C09107=1097.158,375.696,407.850,178.891,20.769,152.741
C09108=1097.152,375.448,407.886,178.888,20.763,152.740
C09109=1097.146,375.200,407.923,178.886,20.758,152.739
C09110=1097.140,374.954,407.959,178.883,20.754,152.739
C09111=1097.134,374.706,407.995,178.880,20.748,152.738
C09112=1097.129,374.459,408.032,178.878,20.743,152.737
C09113=1097.123,374.211,408.068,178.875,20.738,152.736
C09114=1097.118,373.965,408.104,178.872,20.733,152.736
C09115=1097.111,373.718,408.141,178.869,20.728,152.735
C09116=1097.105,373.470,408.177,178.866,20.722,152.734
C09117=1097.099,373.223,408.213,178.863,20.718,152.733
C09118=1097.094,372.976,408.249,178.860,20.712,152.733
C09119=1097.088,372.729,408.286,178.857,20.708,152.732
C09120=1097.082,372.481,408.321,178.855,20.703,152.731
C09121=1097.076,372.234,408.358,178.851,20.698,152.730
C09122=1097.070,371.987,408.393,178.849,20.693,152.730
C09123=1097.065,371.739,408.429,178.845,20.688,152.729
C09124=1097.059,371.492,408.466,178.842,20.683,152.728
C09125=1097.053,371.245,408.501,178.839,20.678,152.728
C09126=1097.047,370.998,408.538,178.836,20.673,152.727
C09127=1097.037,370.603,408.595,178.832,20.665,152.726
C09128=1097.029,370.208,408.652,178.828,20.657,152.725
C09129=1097.019,369.813,408.710,178.823,20.649,152.724
C09130=1097.010,369.418,408.767,178.818,20.642,152.722
C09131=1097.004,369.171,408.802,178.816,20.637,152.722
C09132=1096.999,368.924,408.838,178.812,20.632,152.721
C09133=1096.993,368.677,408.874,178.809,20.628,152.721
C09134=1096.987,368.429,408.910,178.806,20.623,152.720
C09135=1096.982,368.182,408.946,178.803,20.617,152.719
C09136=1096.976,367.934,408.982,178.801,20.613,152.718
C09137=1096.970,367.688,409.018,178.798,20.608,152.718
C09138=1096.964,367.440,409.053,178.795,20.603,152.717
C09139=1096.958,367.192,409.089,178.792,20.599,152.716
C09140=1096.953,366.945,409.125,178.789,20.594,152.716
C09141=1096.947,366.698,409.160,178.786,20.589,152.715
C09142=1096.941,366.451,409.196,178.783,20.585,152.715
C09143=1096.935,366.203,409.231,178.780,20.580,152.714
C09144=1096.930,365.956,409.267,178.777,20.575,152.713
C09145=1096.924,365.708,409.302,178.774,20.570,152.713
C09146=1096.918,365.461,409.338,178.772,20.566,152.712
C09147=1096.912,365.214,409.374,178.769,20.561,152.711
C09148=1096.906,364.966,409.409,178.766,20.556,152.711
C09149=1096.901,364.719,409.445,178.762,20.552,152.710
C09150=1096.895,364.471,409.480,178.760,20.548,152.710
C09151=1096.889,364.224,409.516,178.757,20.543,152.709
C09152=1096.884,363.976,409.551,178.754,20.538,152.708
C09153=1096.878,363.729,409.586,178.750,20.534,152.708
C09154=1096.872,363.482,409.622,178.747,20.529,152.707
C09155=1096.866,363.235,409.657,178.745,20.525,152.707
C09156=1096.860,362.987,409.692,178.742,20.520,152.706
C09157=1096.854,362.740,409.728,178.739,20.515,152.705
C09158=1096.849,362.492,409.763,178.736,20.512,152.705
C09159=1096.843,362.245,409.798,178.733,20.507,152.704
C09160=1096.837,361.997,409.834,178.730,20.502,152.704
C09161=1096.831,361.751,409.869,178.727,20.497,152.703
C09162=1096.825,361.502,409.904,178.724,20.494,152.703
C09163=1096.820,361.255,409.939,178.721,20.489,152.702
C09164=1096.814,361.008,409.975,178.718,20.484,152.701
C09165=1096.809,360.760,410.009,178.714,20.480,152.701
C09166=1096.803,360.513,410.044,178.712,20.476,152.700
C09167=1096.797,360.266,410.080,178.709,20.471,152.700
C09168=1096.791,360.018,410.114,178.706,20.467,152.699
C09169=1096.785,359.770,410.150,178.703,20.463,152.699
C09170=1096.780,359.523,410.184,178.700,20.458,152.698
C09171=1096.774,359.276,410.220,178.697,20.453,152.698
C09172=1096.768,359.029,410.255,178.694,20.450,152.697
C09173=1096.762,358.781,410.290,178.691,20.445,152.697
C09174=1096.756,358.534,410.325,178.688,20.441,152.696
C09175=1096.750,358.286,410.359,178.685,20.437,152.696
C09176=1096.744,358.039,410.395,178.682,20.432,152.695
C09177=1096.739,357.791,410.430,178.679,20.428,152.695
C09178=1096.732,357.544,410.465,178.676,20.424,152.694
C09179=1096.724,357.164,410.517,178.671,20.417,152.693
C09180=1096.716,356.784,410.572,178.667,20.410,152.692
C09181=1096.707,356.405,410.625,178.662,20.404,152.692
C09182=1096.698,356.025,410.678,178.658,20.398,152.691
C09183=1096.692,355.778,410.713,178.654,20.393,152.690
C09184=1096.686,355.530,410.748,178.652,20.389,152.690
C09185=1096.681,355.282,410.782,178.648,20.385,152.689
C09186=1096.675,355.035,410.817,178.645,20.381,152.689
C09187=1096.669,354.787,410.852,178.643,20.377,152.688
C09188=1096.663,354.540,410.886,178.639,20.372,152.688
C09189=1096.658,354.292,410.921,178.637,20.369,152.687
C09190=1096.652,354.044,410.955,178.634,20.364,152.687
C09191=1096.646,353.797,410.991,178.630,20.360,152.687
C09192=1096.640,353.550,411.025,178.628,20.356,152.686
C09193=1096.635,353.302,411.059,178.624,20.352,152.686
C09194=1096.629,353.054,411.094,178.621,20.348,152.685
C09195=1096.624,352.807,411.128,178.618,20.344,152.685
C09196=1096.618,352.560,411.162,178.615,20.339,152.684
C09197=1096.611,352.312,411.197,178.612,20.336,152.684
C09198=1096.606,352.065,411.232,178.609,20.331,152.683
C09199=1096.600,351.817,411.266,178.606,20.328,152.683
C09200=1096.594,351.570,411.300,178.603,20.324,152.682
C09201=1096.588,351.322,411.335,178.600,20.320,152.682
C09202=1096.583,351.074,411.369,178.597,20.316,152.682
C09203=1096.577,350.827,411.403,178.594,20.312,152.681
C09204=1096.572,350.580,411.438,178.591,20.308,152.681
C09205=1096.565,350.332,411.473,178.588,20.304,152.680
C09206=1096.559,350.084,411.507,178.584,20.299,152.680
C09207=1096.554,349.837,411.541,178.582,20.296,152.679
C09208=1096.549,349.589,411.575,178.578,20.292,152.679
C09209=1096.542,349.341,411.609,178.576,20.288,152.679
C09210=1096.537,349.093,411.644,178.572,20.284,152.678
C09211=1096.531,348.846,411.678,178.570,20.280,152.678
C09212=1096.525,348.599,411.712,178.566,20.276,152.677
C09213=1096.519,348.351,411.746,178.564,20.273,152.677
C09214=1096.514,348.103,411.781,178.560,20.269,152.677
C09215=1096.508,347.855,411.814,178.557,20.264,152.676
C09216=1096.502,347.608,411.848,178.554,20.261,152.676
C09217=1096.496,347.361,411.882,178.551,20.257,152.675
C09218=1096.491,347.113,411.917,178.548,20.253,152.675
C09219=1096.486,346.865,411.950,178.545,20.249,152.675
C09220=1096.480,346.618,411.984,178.542,20.245,152.674
C09221=1096.473,346.370,412.019,178.539,20.241,152.674
C09222=1096.468,346.123,412.053,178.536,20.238,152.673
C09223=1096.463,345.874,412.087,178.532,20.234,152.673
C09224=1096.457,345.627,412.121,178.530,20.230,152.673
C09225=1096.451,345.379,412.154,178.527,20.226,152.672
C09226=1096.445,345.132,412.188,178.524,20.222,152.672
C09227=1096.440,344.885,412.222,178.520,20.218,152.671
C09228=1096.434,344.637,412.256,178.518,20.215,152.671
C09229=1096.428,344.389,412.290,178.514,20.211,152.671
C09230=1096.422,344.141,412.323,178.512,20.207,152.670
C09231=1096.413,343.764,412.375,178.507,20.202,152.670
C09232=1096.405,343.387,412.427,178.502,20.196,152.669
C09233=1096.396,343.009,412.478,178.497,20.190,152.669
C09234=1096.387,342.632,412.529,178.492,20.185,152.668
C09235=1096.381,342.385,412.563,178.489,20.181,152.668
C09236=1096.376,342.137,412.596,178.487,20.178,152.668
C09237=1096.370,341.890,412.630,178.483,20.174,152.667
C09238=1096.365,341.642,412.664,178.481,20.170,152.667
C09239=1096.359,341.394,412.698,178.477,20.167,152.667
C09240=1096.353,341.147,412.731,178.474,20.163,152.666
C09241=1096.347,340.898,412.765,178.471,20.159,152.666
C09242=1096.341,340.651,412.799,178.468,20.156,152.666
C09243=1096.336,340.403,412.832,178.465,20.152,152.665
C09244=1096.330,340.155,412.865,178.462,20.149,152.665
C09245=1096.324,339.907,412.899,178.458,20.145,152.665
C09246=1096.318,339.660,412.932,178.455,20.141,152.664
C09247=1096.312,339.412,412.966,178.453,20.138,152.664
C09248=1096.307,339.165,412.999,178.449,20.134,152.664
C09249=1096.302,338.917,413.032,178.446,20.131,152.663
C09250=1096.296,338.670,413.066,178.443,20.127,152.663
C09251=1096.290,338.422,413.099,178.440,20.124,152.663
C09252=1096.285,338.174,413.133,178.437,20.120,152.662
C09253=1096.278,337.926,413.165,178.434,20.116,152.662
C09254=1096.273,337.678,413.199,178.431,20.113,152.662
C09255=1096.267,337.430,413.232,178.427,20.109,152.662
C09256=1096.262,337.183,413.266,178.425,20.106,152.661
C09257=1096.255,336.936,413.299,178.421,20.102,152.661
C09258=1096.250,336.688,413.332,178.418,20.099,152.661
C09259=1096.244,336.440,413.365,178.415,20.096,152.660
C09260=1096.239,336.192,413.399,178.412,20.092,152.660
C09261=1096.232,335.944,413.432,178.409,20.089,152.660
C09262=1096.227,335.696,413.465,178.405,20.085,152.660
C09263=1096.221,335.448,413.498,178.403,20.082,152.659
C09264=1096.215,335.201,413.531,178.400,20.079,152.659
C09265=1096.209,334.953,413.564,178.396,20.075,152.659
C09266=1096.204,334.705,413.598,178.393,20.072,152.658
C09267=1096.198,334.457,413.631,178.391,20.069,152.658
C09268=1096.193,334.210,413.663,178.387,20.064,152.658
C09269=1096.187,333.962,413.697,178.384,20.061,152.658
C09270=1096.181,333.714,413.730,178.382,20.058,152.657
C09271=1096.175,333.466,413.762,178.378,20.054,152.657
C09272=1096.170,333.218,413.795,178.375,20.051,152.657
C09273=1096.164,332.971,413.828,178.371,20.047,152.657
C09274=1096.158,332.723,413.861,178.369,20.044,152.656
C09275=1096.153,332.476,413.894,178.366,20.041,152.656
C09276=1096.147,332.228,413.927,178.362,20.038,152.656
C09277=1096.142,331.979,413.960,178.359,20.034,152.656
C09278=1096.135,331.732,413.993,178.356,20.031,152.655
C09279=1096.130,331.484,414.026,178.353,20.027,152.655
C09280=1096.123,331.236,414.059,178.350,20.024,152.655
C09281=1096.118,330.988,414.091,178.347,20.021,152.655
C09282=1096.112,330.740,414.124,178.343,20.018,152.654
C09283=1096.103,330.358,414.174,178.339,20.013,152.654
C09284=1096.094,329.974,414.225,178.334,20.008,152.654
C09285=1096.085,329.591,414.276,178.329,20.003,152.653
C09286=1096.076,329.208,414.326,178.324,19.998,152.653
C09287=1096.070,328.960,414.359,178.321,19.995,152.653
C09288=1096.064,328.712,414.391,178.318,19.992,152.653
C09289=1096.059,328.464,414.424,178.315,19.989,152.653
C09290=1096.053,328.216,414.456,178.312,19.986,152.652
C09291=1096.047,327.969,414.489,178.308,19.982,152.652
C09292=1096.042,327.721,414.521,178.305,19.979,152.652
C09293=1096.035,327.473,414.554,178.303,19.976,152.652
C09294=1096.029,327.225,414.586,178.299,19.973,152.652
C09295=1096.024,326.978,414.619,178.296,19.970,152.651
C09296=1096.019,326.729,414.651,178.293,19.967,152.651
C09297=1096.012,326.482,414.684,178.290,19.964,152.651
C09298=1096.006,326.234,414.716,178.286,19.960,152.651
C09299=1096.001,325.986,414.749,178.283,19.957,152.651
C09300=1095.995,325.738,414.781,178.281,19.954,152.650
C09301=1095.989,325.491,414.814,178.278,19.951,152.650
C09302=1095.983,325.242,414.846,178.274,19.948,152.650
C09303=1095.978,324.994,414.878,178.271,19.945,152.650
C09304=1095.972,324.747,414.911,178.268,19.942,152.650
C09305=1095.966,324.499,414.943,178.265,19.939,152.649
C09306=1095.961,324.251,414.974,178.261,19.935,152.649
C09307=1095.955,324.003,415.008,178.258,19.932,152.649
C09308=1095.949,323.755,415.040,178.255,19.929,152.649
C09309=1095.944,323.508,415.071,178.253,19.926,152.649
C09310=1095.938,323.259,415.103,178.249,19.923,152.648
C09311=1095.933,323.012,415.136,178.246,19.920,152.648
C09312=1095.927,322.764,415.168,178.243,19.917,152.648
C09313=1095.921,322.516,415.200,178.240,19.914,152.648
C09314=1095.915,322.268,415.232,178.236,19.910,152.648
C09315=1095.909,322.020,415.264,178.233,19.908,152.648
C09316=1095.903,321.772,415.297,178.230,19.905,152.647
C09317=1095.899,321.525,415.329,178.227,19.902,152.647
C09318=1095.893,321.276,415.361,178.223,19.899,152.647
C09319=1095.887,321.029,415.393,178.221,19.895,152.647
C09320=1095.881,320.781,415.425,178.218,19.892,152.647
C09321=1095.876,320.533,415.457,178.215,19.890,152.647
C09322=1095.870,320.285,415.489,178.212,19.887,152.646
C09323=1095.864,320.037,415.520,178.208,19.883,152.646
C09324=1095.859,319.789,415.554,178.205,19.881,152.646
C09325=1095.853,319.541,415.586,178.202,19.877,152.646
C09326=1095.848,319.294,415.617,178.199,19.874,152.646
C09327=1095.842,319.046,415.649,178.196,19.872,152.646
C09328=1095.836,318.798,415.681,178.192,19.868,152.645
C09329=1095.830,318.550,415.713,178.190,19.865,152.645
C09330=1095.825,318.302,415.745,178.186,19.863,152.645
C09331=1095.820,318.054,415.776,178.184,19.860,152.645
C09332=1095.814,317.806,415.808,178.180,19.857,152.645
C09333=1095.808,317.558,415.839,178.177,19.853,152.645
C09334=1095.803,317.310,415.872,178.174,19.850,152.644
C09335=1095.794,316.920,415.922,178.169,19.846,152.644
C09336=1095.785,316.529,415.971,178.164,19.841,152.644
C09337=1095.776,316.139,416.022,178.159,19.836,152.644
C09338=1095.768,315.749,416.071,178.154,19.832,152.644
C09339=1095.762,315.501,416.103,178.151,19.829,152.643
C09340=1095.756,315.254,416.135,178.148,19.826,152.643
C09341=1095.751,315.006,416.166,178.145,19.823,152.643
C09342=1095.745,314.758,416.198,178.142,19.820,152.643
C09343=1095.740,314.510,416.229,178.138,19.818,152.643
C09344=1095.733,314.262,416.261,178.135,19.815,152.643
C09345=1095.728,314.014,416.292,178.132,19.812,152.643
C09346=1095.722,313.765,416.324,178.129,19.809,152.643
C09347=1095.716,313.518,416.355,178.125,19.806,152.643
C09348=1095.710,313.270,416.387,178.122,19.804,152.643
C09349=1095.705,313.022,416.418,178.119,19.801,152.642
C09350=1095.698,312.774,416.449,178.116,19.798,152.642
C09351=1095.693,312.526,416.481,178.113,19.796,152.642
C09352=1095.687,312.278,416.512,178.110,19.793,152.642
C09353=1095.681,312.030,416.543,178.107,19.790,152.642
C09354=1095.675,311.782,416.575,178.104,19.787,152.642
C09355=1095.670,311.534,416.606,178.100,19.784,152.642
C09356=1095.664,311.287,416.637,178.097,19.782,152.642
C09357=1095.658,311.038,416.668,178.094,19.779,152.642
C09358=1095.653,310.790,416.700,178.091,19.776,152.642
C09359=1095.646,310.542,416.731,178.088,19.774,152.642
C09360=1095.641,310.294,416.763,178.085,19.771,152.641
C09361=1095.635,310.047,416.793,178.082,19.768,152.641
C09362=1095.629,309.798,416.825,178.079,19.766,152.641
C09363=1095.624,309.550,416.856,178.075,19.762,152.641
C09364=1095.618,309.303,416.887,178.072,19.760,152.641
C09365=1095.612,309.054,416.918,178.068,19.757,152.641
C09366=1095.606,308.807,416.949,178.065,19.755,152.641
C09367=1095.601,308.559,416.980,178.062,19.752,152.641
C09368=1095.594,308.311,417.012,178.059,19.749,152.641
C09369=1095.589,308.063,417.043,178.056,19.747,152.641
C09370=1095.583,307.815,417.073,178.053,19.744,152.641
C09371=1095.578,307.568,417.105,178.050,19.741,152.641
C09372=1095.572,307.319,417.136,178.046,19.738,152.641
C09373=1095.566,307.071,417.166,178.043,19.736,152.641
C09374=1095.561,306.823,417.198,178.040,19.733,152.641
C09375=1095.555,306.576,417.228,178.037,19.730,152.640
C09376=1095.550,306.327,417.260,178.034,19.728,152.640
C09377=1095.544,306.079,417.290,178.030,19.725,152.640
C09378=1095.538,305.831,417.322,178.027,19.723,152.640
C09379=1095.533,305.584,417.352,178.024,19.720,152.640
C09380=1095.527,305.335,417.383,178.021,19.717,152.640
C09381=1095.521,305.087,417.414,178.017,19.714,152.640
C09382=1095.515,304.840,417.445,178.014,19.712,152.640
C09383=1095.510,304.592,417.476,178.011,19.709,152.640
C09384=1095.504,304.344,417.506,178.008,19.706,152.640
C09385=1095.499,304.096,417.537,178.005,19.704,152.640
C09386=1095.493,303.847,417.568,178.002,19.701,152.640
C09387=1095.485,303.460,417.616,177.997,19.697,152.640
C09388=1095.475,303.072,417.664,177.992,19.693,152.640
C09389=1095.467,302.685,417.712,177.987,19.689,152.639
C09390=1095.458,302.296,417.760,177.982,19.685,152.639
C09391=1095.453,302.048,417.791,177.979,19.682,152.639
C09392=1095.447,301.800,417.821,177.975,19.679,152.639
C09393=1095.441,301.553,417.852,177.972,19.676,152.639
C09394=1095.436,301.305,417.883,177.969,19.674,152.639
C09395=1095.430,301.057,417.913,177.966,19.671,152.639
C09396=1095.424,300.809,417.943,177.963,19.669,152.639
C09397=1095.419,300.561,417.974,177.960,19.666,152.639
C09398=1095.413,300.313,418.004,177.957,19.663,152.639
C09399=1095.408,300.065,418.035,177.953,19.661,152.639
C09400=1095.402,299.817,418.065,177.950,19.659,152.639
C09401=1095.397,299.569,418.096,177.947,19.656,152.639
C09402=1095.392,299.321,418.127,177.944,19.653,152.639
C09403=1095.386,299.073,418.157,177.941,19.651,152.639
C09404=1095.379,298.825,418.188,177.938,19.648,152.639
C09405=1095.375,298.576,418.218,177.935,19.645,152.639
C09406=1095.369,298.328,418.248,177.932,19.643,152.639
C09407=1095.363,298.080,418.279,177.928,19.641,152.639
C09408=1095.357,297.832,418.309,177.925,19.638,152.639
C09409=1095.352,297.584,418.339,177.922,19.635,152.639
C09410=1095.347,297.336,418.370,177.919,19.633,152.639
C09411=1095.341,297.088,418.400,177.916,19.631,152.639
C09412=1095.335,296.840,418.430,177.913,19.628,152.639
C09413=1095.329,296.592,418.460,177.910,19.625,152.638
C09414=1095.324,296.344,418.490,177.906,19.623,152.639
C09415=1095.318,296.096,418.521,177.903,19.621,152.638
C09416=1095.312,295.848,418.550,177.900,19.618,152.638
C09417=1095.306,295.600,418.581,177.897,19.616,152.638
C09418=1095.301,295.352,418.611,177.894,19.613,152.638
C09419=1095.295,295.104,418.641,177.890,19.611,152.639
C09420=1095.289,294.856,418.671,177.887,19.608,152.638
C09421=1095.283,294.608,418.701,177.884,19.606,152.638
C09422=1095.278,294.360,418.731,177.881,19.604,152.638
C09423=1095.272,294.112,418.761,177.878,19.601,152.638
C09424=1095.267,293.863,418.791,177.874,19.599,152.639
C09425=1095.261,293.615,418.821,177.871,19.596,152.638
C09426=1095.255,293.367,418.851,177.868,19.594,152.638
C09427=1095.249,293.119,418.881,177.865,19.591,152.638
C09428=1095.244,292.871,418.911,177.862,19.589,152.638
C09429=1095.238,292.623,418.941,177.859,19.587,152.638
C09430=1095.233,292.374,418.971,177.855,19.584,152.638
C09431=1095.227,292.127,419.001,177.852,19.582,152.639
C09432=1095.221,291.878,419.031,177.849,19.579,152.638
C09433=1095.215,291.630,419.061,177.846,19.577,152.639
C09434=1095.210,291.382,419.091,177.843,19.574,152.638
C09435=1095.204,291.134,419.121,177.839,19.572,152.639
C09436=1095.199,290.886,419.151,177.836,19.570,152.639
C09437=1095.194,290.638,419.180,177.833,19.567,152.639
C09438=1095.188,290.390,419.211,177.830,19.565,152.639
C09439=1095.179,290.016,419.255,177.825,19.561,152.639
C09440=1095.170,289.643,419.300,177.820,19.558,152.639
C09441=1095.162,289.268,419.345,177.815,19.554,152.639
C09442=1095.154,288.895,419.389,177.811,19.550,152.639
C09443=1095.148,288.647,419.419,177.807,19.548,152.639
C09444=1095.142,288.399,419.448,177.804,19.546,152.639
C09445=1095.136,288.151,419.478,177.801,19.543,152.639
C09446=1095.131,287.902,419.508,177.797,19.541,152.639
C09447=1095.125,287.654,419.537,177.795,19.539,152.639
C09448=1095.119,287.406,419.566,177.792,19.537,152.639
C09449=1095.113,287.158,419.597,177.789,19.535,152.639
C09450=1095.108,286.909,419.626,177.785,19.532,152.639
C09451=1095.102,286.662,419.655,177.782,19.530,152.639
C09452=1095.096,286.413,419.685,177.779,19.527,152.639
C09453=1095.091,286.165,419.714,177.776,19.525,152.639
C09454=1095.085,285.917,419.744,177.772,19.523,152.639
C09455=1095.079,285.668,419.773,177.769,19.521,152.639
C09456=1095.074,285.420,419.803,177.766,19.518,152.639
C09457=1095.069,285.172,419.832,177.763,19.516,152.639
C09458=1095.062,284.925,419.862,177.760,19.514,152.639
C09459=1095.057,284.676,419.891,177.756,19.511,152.639
C09460=1095.051,284.428,419.921,177.753,19.509,152.639
C09461=1095.045,284.180,419.950,177.751,19.507,152.639
C09462=1095.040,283.932,419.979,177.747,19.505,152.639
C09463=1095.035,283.683,420.008,177.744,19.503,152.639
C09464=1095.029,283.435,420.037,177.741,19.500,152.639
C09465=1095.023,283.186,420.067,177.738,19.498,152.639
C09466=1095.017,282.939,420.095,177.734,19.496,152.640
C09467=1095.012,282.691,420.125,177.731,19.493,152.640
C09468=1095.006,282.442,420.155,177.728,19.491,152.640
C09469=1095.000,282.194,420.184,177.724,19.489,152.640
C09470=1094.995,281.946,420.213,177.721,19.486,152.640
C09471=1094.989,281.698,420.242,177.719,19.485,152.640
C09472=1094.983,281.450,420.272,177.716,19.482,152.640
C09473=1094.978,281.201,420.301,177.712,19.480,152.640
C09474=1094.973,280.953,420.329,177.709,19.478,152.640
C09475=1094.967,280.705,420.359,177.706,19.475,152.640
C09476=1094.961,280.457,420.388,177.702,19.473,152.640
C09477=1094.955,280.209,420.417,177.699,19.471,152.640
C09478=1094.950,279.960,420.446,177.696,19.469,152.640
C09479=1094.944,279.712,420.475,177.693,19.466,152.640
C09480=1094.938,279.463,420.504,177.690,19.465,152.640
C09481=1094.933,279.216,420.533,177.687,19.463,152.640
C09482=1094.927,278.967,420.562,177.684,19.460,152.640
C09483=1094.921,278.719,420.591,177.681,19.458,152.640
C09484=1094.916,278.471,420.620,177.677,19.456,152.640
C09485=1094.910,278.222,420.648,177.674,19.453,152.641
C09486=1094.904,277.974,420.678,177.671,19.451,152.641
C09487=1094.899,277.727,420.707,177.668,19.449,152.641
C09488=1094.893,277.478,420.735,177.665,19.447,152.641
C09489=1094.888,277.229,420.765,177.662,19.445,152.641
C09490=1094.882,276.981,420.793,177.658,19.443,152.641
C09491=1094.874,276.617,420.836,177.653,19.439,152.641
C09492=1094.865,276.253,420.878,177.649,19.436,152.641
C09493=1094.857,275.888,420.920,177.644,19.433,152.641
C09494=1094.849,275.524,420.962,177.639,19.430,152.641
C09495=1094.843,275.276,420.990,177.636,19.428,152.641
C09496=1094.838,275.027,421.020,177.634,19.426,152.641
C09497=1094.832,274.779,421.048,177.630,19.424,152.642
C09498=1094.826,274.531,421.077,177.627,19.422,152.642
C09499=1094.821,274.283,421.105,177.624,19.419,152.642
C09500=1094.815,274.034,421.134,177.621,19.417,152.642
C09501=1094.809,273.786,421.163,177.617,19.415,152.642
C09502=1094.804,273.538,421.191,177.615,19.413,152.642
C09503=1094.798,273.289,421.220,177.611,19.411,152.642
C09504=1094.793,273.041,421.248,177.608,19.409,152.642
C09505=1094.787,272.793,421.277,177.605,19.406,152.642
C09506=1094.781,272.544,421.306,177.601,19.404,152.642
C09507=1094.775,272.296,421.334,177.598,19.402,152.642
C09508=1094.769,272.048,421.363,177.596,19.400,152.642
C09509=1094.765,271.800,421.391,177.592,19.398,152.642
C09510=1094.759,271.551,421.420,177.589,19.396,152.643
C09511=1094.753,271.303,421.447,177.586,19.394,152.643
C09512=1094.747,271.055,421.477,177.582,19.392,152.643
C09513=1094.742,270.807,421.504,177.579,19.390,152.643
C09514=1094.736,270.558,421.533,177.576,19.388,152.643
C09515=1094.730,270.309,421.561,177.573,19.385,152.643
C09516=1094.724,270.062,421.590,177.570,19.383,152.643
C09517=1094.719,269.813,421.619,177.567,19.381,152.643
C09518=1094.714,269.565,421.647,177.563,19.379,152.643
C09519=1094.708,269.316,421.675,177.561,19.377,152.643
C09520=1094.702,269.068,421.703,177.558,19.375,152.643
C09521=1094.696,268.819,421.731,177.554,19.373,152.643
C09522=1094.691,268.572,421.760,177.551,19.371,152.644
C09523=1094.685,268.323,421.788,177.547,19.369,152.644
C09524=1094.679,268.075,421.816,177.545,19.367,152.644
C09525=1094.674,267.826,421.845,177.542,19.365,152.644
C09526=1094.668,267.578,421.873,177.538,19.363,152.644
C09527=1094.662,267.329,421.901,177.535,19.361,152.644
C09528=1094.657,267.081,421.929,177.532,19.359,152.644
C09529=1094.652,266.833,421.957,177.529,19.357,152.644
C09530=1094.646,266.584,421.985,177.526,19.355,152.644
C09531=1094.640,266.336,422.013,177.522,19.353,152.645
C09532=1094.634,266.088,422.041,177.519,19.351,152.645
C09533=1094.629,265.840,422.069,177.516,19.348,152.645
C09534=1094.623,265.591,422.098,177.513,19.347,152.645
C09535=1094.618,265.343,422.126,177.510,19.345,152.645
C09536=1094.612,265.095,422.153,177.507,19.342,152.645
C09537=1094.606,264.846,422.181,177.503,19.340,152.645
C09538=1094.600,264.598,422.209,177.501,19.339,152.645
C09539=1094.595,264.349,422.237,177.497,19.336,152.645
C09540=1094.589,264.101,422.265,177.494,19.334,152.645
C09541=1094.583,263.852,422.293,177.491,19.333,152.646
C09542=1094.577,263.604,422.321,177.488,19.331,152.646
C09543=1094.570,263.243,422.362,177.483,19.328,152.646
C09544=1094.561,262.880,422.402,177.479,19.325,152.646
C09545=1094.553,262.519,422.443,177.474,19.322,152.646
C09546=1094.544,262.158,422.483,177.470,19.319,152.646
C09547=1094.538,261.910,422.510,177.466,19.317,152.647
C09548=1094.532,261.661,422.538,177.463,19.315,152.647
C09549=1094.527,261.413,422.566,177.459,19.313,152.647
C09550=1094.520,261.164,422.594,177.457,19.312,152.647
C09551=1094.515,260.916,422.621,177.453,19.310,152.647
C09552=1094.510,260.668,422.649,177.450,19.307,152.647
C09553=1094.503,260.419,422.677,177.447,19.306,152.647
C09554=1094.498,260.170,422.704,177.444,19.304,152.647
C09555=1094.493,259.922,422.732,177.441,19.302,152.648
C09556=1094.486,259.674,422.760,177.437,19.300,152.648
C09557=1094.481,259.425,422.787,177.434,19.298,152.648
C09558=1094.475,259.177,422.815,177.431,19.296,152.648
C09559=1094.470,258.928,422.842,177.428,19.294,152.648
C09560=1094.464,258.680,422.870,177.425,19.292,152.648
C09561=1094.458,258.432,422.898,177.422,19.290,152.648
C09562=1094.453,258.183,422.925,177.419,19.288,152.648
C09563=1094.447,257.935,422.953,177.415,19.287,152.649
C09564=1094.441,257.687,422.980,177.412,19.284,152.649
C09565=1094.435,257.438,423.008,177.410,19.283,152.649
C09566=1094.430,257.190,423.034,177.406,19.281,152.649
C09567=1094.424,256.941,423.062,177.403,19.279,152.649
C09568=1094.419,256.692,423.090,177.399,19.277,152.649
C09569=1094.413,256.444,423.117,177.397,19.275,152.649
C09570=1094.408,256.196,423.145,177.393,19.273,152.649
C09571=1094.402,255.948,423.172,177.390,19.271,152.650
C09572=1094.396,255.699,423.200,177.387,19.270,152.650
C09573=1094.390,255.450,423.226,177.384,19.267,152.650
C09574=1094.385,255.202,423.254,177.381,19.265,152.650
C09575=1094.380,254.954,423.281,177.377,19.263,152.650
C09576=1094.374,254.706,423.309,177.375,19.262,152.650
C09577=1094.368,254.456,423.336,177.371,19.260,152.650
C09578=1094.362,254.208,423.363,177.368,19.258,152.651
C09579=1094.357,253.960,423.391,177.366,19.256,152.651
C09580=1094.351,253.712,423.418,177.362,19.254,152.651
C09581=1094.346,253.463,423.445,177.359,19.252,152.651
C09582=1094.340,253.214,423.472,177.355,19.250,152.651
C09583=1094.334,252.966,423.500,177.353,19.248,152.651
C09584=1094.329,252.717,423.527,177.350,19.246,152.651
C09585=1094.324,252.469,423.554,177.346,19.244,152.651
C09586=1094.318,252.220,423.580,177.343,19.243,152.652
C09587=1094.312,251.972,423.608,177.340,19.241,152.652
C09588=1094.306,251.723,423.635,177.337,19.238,152.652
C09589=1094.301,251.475,423.663,177.334,19.237,152.652
C09590=1094.295,251.226,423.689,177.331,19.235,152.652
C09591=1094.289,250.978,423.716,177.327,19.233,152.652
C09592=1094.284,250.729,423.743,177.325,19.231,152.652
C09593=1094.278,250.482,423.771,177.322,19.229,152.652
C09594=1094.273,250.233,423.798,177.318,19.227,152.653
C09595=1094.265,249.868,423.837,177.314,19.224,152.653
C09596=1094.257,249.504,423.877,177.309,19.222,152.653
C09597=1094.249,249.139,423.917,177.305,19.219,152.653
C09598=1094.241,248.775,423.955,177.301,19.216,152.653
C09599=1094.235,248.526,423.983,177.297,19.214,152.654
C09600=1094.229,248.277,424.010,177.294,19.212,152.654
C09601=1094.224,248.029,424.036,177.291,19.211,152.654
C09602=1094.219,247.780,424.064,177.288,19.208,152.654
C09603=1094.213,247.532,424.090,177.285,19.206,152.654
C09604=1094.208,247.283,424.118,177.282,19.205,152.654
C09605=1094.202,247.035,424.144,177.278,19.203,152.654
C09606=1094.196,246.786,424.171,177.275,19.201,152.654
C09607=1094.190,246.538,424.197,177.272,19.200,152.655
C09608=1094.185,246.290,424.224,177.269,19.197,152.655
C09609=1094.180,246.041,424.251,177.266,19.195,152.655
C09610=1094.174,245.793,424.278,177.263,19.194,152.655
C09611=1094.168,245.544,424.304,177.260,19.192,152.655
C09612=1094.163,245.295,424.331,177.256,19.190,152.655
C09613=1094.158,245.047,424.358,177.254,19.188,152.655
C09614=1094.152,244.798,424.384,177.250,19.186,152.656
C09615=1094.146,244.550,424.411,177.247,19.184,152.656
C09616=1094.140,244.302,424.438,177.245,19.183,152.656
C09617=1094.135,244.053,424.464,177.241,19.181,152.656
C09618=1094.129,243.804,424.490,177.238,19.179,152.656
C09619=1094.124,243.556,424.518,177.235,19.177,152.656
C09620=1094.118,243.307,424.544,177.232,19.175,152.656
C09621=1094.113,243.058,424.570,177.228,19.173,152.657
C09622=1094.107,242.810,424.597,177.226,19.172,152.657
C09623=1094.101,242.562,424.623,177.222,19.170,152.657
C09624=1094.095,242.313,424.650,177.220,19.168,152.657
C09625=1094.090,242.064,424.676,177.216,19.166,152.657
C09626=1094.084,241.816,424.703,177.213,19.164,152.657
C09627=1094.078,241.567,424.729,177.210,19.163,152.658
C09628=1094.073,241.319,424.755,177.207,19.161,152.658
C09629=1094.067,241.070,424.782,177.203,19.159,152.658
C09630=1094.061,240.822,424.809,177.201,19.157,152.658
C09631=1094.056,240.573,424.835,177.197,19.156,152.658
C09632=1094.050,240.324,424.861,177.195,19.154,152.658
C09633=1094.045,240.075,424.887,177.191,19.152,152.659
C09634=1094.039,239.827,424.914,177.188,19.150,152.659
C09635=1094.033,239.578,424.940,177.185,19.148,152.659
C09636=1094.028,239.330,424.966,177.182,19.147,152.659
C09637=1094.022,239.081,424.993,177.179,19.145,152.659
C09638=1094.016,238.832,425.019,177.176,19.143,152.659
C09639=1094.011,238.585,425.045,177.173,19.141,152.659
C09640=1094.006,238.336,425.071,177.170,19.140,152.660
C09641=1093.999,238.088,425.097,177.166,19.138,152.660
C09642=1093.994,237.839,425.123,177.164,19.136,152.660
C09643=1093.988,237.590,425.149,177.160,19.135,152.660
C09644=1093.982,237.341,425.176,177.157,19.132,152.660
C09645=1093.977,237.092,425.202,177.155,19.131,152.660
C09646=1093.971,236.844,425.228,177.151,19.129,152.661
C09647=1093.963,236.473,425.267,177.147,19.126,152.661
C09648=1093.954,236.102,425.306,177.142,19.124,152.661
C09649=1093.946,235.730,425.345,177.137,19.121,152.661
C09650=1093.938,235.359,425.383,177.133,19.119,152.662
C09651=1093.933,235.110,425.410,177.130,19.117,152.662
C09652=1093.927,234.861,425.436,177.127,19.115,152.662
C09653=1093.921,234.613,425.461,177.124,19.113,152.662
C09654=1093.916,234.365,425.488,177.120,19.111,152.662
C09655=1093.910,234.116,425.514,177.118,19.110,152.662
C09656=1093.905,233.867,425.540,177.114,19.108,152.662
C09657=1093.899,233.618,425.565,177.112,19.107,152.663
C09658=1093.893,233.370,425.592,177.108,19.104,152.663
C09659=1093.888,233.122,425.617,177.105,19.103,152.663
C09660=1093.882,232.873,425.643,177.102,19.101,152.663
C09661=1093.877,232.624,425.669,177.099,19.099,152.663
C09662=1093.871,232.375,425.694,177.096,19.098,152.664
C09663=1093.865,232.127,425.721,177.093,19.096,152.664
C09664=1093.860,231.878,425.746,177.090,19.094,152.664
C09665=1093.854,231.630,425.772,177.087,19.092,152.664
C09666=1093.848,231.381,425.798,177.084,19.091,152.664
C09667=1093.843,231.132,425.824,177.081,19.089,152.664
C09668=1093.837,230.884,425.849,177.077,19.087,152.665
C09669=1093.832,230.635,425.875,177.075,19.086,152.665
C09670=1093.826,230.386,425.901,177.071,19.083,152.665
C09671=1093.820,230.138,425.927,177.069,19.082,152.665
C09672=1093.815,229.889,425.952,177.065,19.080,152.665
C09673=1093.809,229.641,425.977,177.062,19.079,152.665
C09674=1093.803,229.392,426.003,177.059,19.077,152.666
C09675=1093.798,229.143,426.029,177.056,19.076,152.666
C09676=1093.792,228.895,426.054,177.053,19.073,152.666
C09677=1093.787,228.646,426.080,177.050,19.072,152.666
C09678=1093.781,228.397,426.106,177.047,19.070,152.666
C09679=1093.775,228.148,426.132,177.043,19.068,152.666
C09680=1093.770,227.900,426.157,177.041,19.067,152.667
C09681=1093.764,227.651,426.182,177.037,19.065,152.667
C09682=1093.758,227.403,426.208,177.035,19.063,152.667
C09683=1093.753,227.154,426.233,177.031,19.062,152.667
C09684=1093.747,226.905,426.258,177.029,19.060,152.667
C09685=1093.742,226.656,426.284,177.025,19.058,152.668
C09686=1093.735,226.407,426.309,177.023,19.057,152.668
C09687=1093.731,226.159,426.335,177.019,19.055,152.668
C09688=1093.724,225.910,426.360,177.017,19.053,152.668
C09689=1093.719,225.662,426.386,177.013,19.052,152.668
C09690=1093.713,225.413,426.411,177.011,19.050,152.668
C09691=1093.707,225.164,426.436,177.007,19.048,152.669
C09692=1093.703,224.916,426.461,177.005,19.047,152.669
C09693=1093.696,224.667,426.487,177.001,19.045,152.669
C09694=1093.691,224.418,426.513,176.999,19.044,152.669
C09695=1093.685,224.170,426.537,176.995,19.042,152.669
C09696=1093.680,223.921,426.563,176.992,19.040,152.669
C09697=1093.674,223.673,426.588,176.989,19.038,152.670
C09698=1093.669,223.424,426.614,176.986,19.037,152.670
C09699=1093.660,223.044,426.652,176.981,19.034,152.670
C09700=1093.652,222.664,426.690,176.977,19.031,152.670
C09701=1093.643,222.284,426.729,176.972,19.029,152.671
C09702=1093.634,221.904,426.768,176.967,19.026,152.671
C09703=1093.629,221.655,426.792,176.965,19.025,152.671
C09704=1093.623,221.406,426.817,176.961,19.023,152.671
C09705=1093.618,221.158,426.843,176.959,19.021,152.671
C09706=1093.612,220.909,426.867,176.955,19.020,152.672
C09707=1093.606,220.660,426.893,176.953,19.019,152.672
C09708=1093.601,220.412,426.917,176.949,19.016,152.672
C09709=1093.595,220.163,426.943,176.946,19.015,152.672
C09710=1093.590,219.915,426.968,176.943,19.013,152.672
C09711=1093.584,219.665,426.992,176.940,19.012,152.673
C09712=1093.578,219.417,427.018,176.937,19.010,152.673
C09713=1093.572,219.168,427.042,176.934,19.009,152.673
C09714=1093.567,218.919,427.068,176.931,19.006,152.673
C09715=1093.561,218.671,427.092,176.928,19.005,152.673
C09716=1093.555,218.422,427.118,176.925,19.003,152.673
C09717=1093.550,218.173,427.142,176.922,19.002,152.674
C09718=1093.544,217.925,427.167,176.919,19.000,152.674
C09719=1093.539,217.676,427.192,176.916,18.999,152.674
C09720=1093.533,217.426,427.217,176.913,18.998,152.674
C09721=1093.528,217.179,427.242,176.910,18.995,152.674
C09722=1093.522,216.929,427.266,176.907,18.994,152.675
C09723=1093.516,216.681,427.291,176.904,18.992,152.675
C09724=1093.510,216.432,427.316,176.901,18.991,152.675
C09725=1093.505,216.183,427.340,176.898,18.989,152.675
C09726=1093.500,215.934,427.366,176.895,18.988,152.675
C09727=1093.494,215.686,427.390,176.892,18.985,152.675
C09728=1093.489,215.438,427.415,176.889,18.984,152.676
C09729=1093.483,215.189,427.440,176.886,18.982,152.676
C09730=1093.477,214.940,427.464,176.883,18.981,152.676
C09731=1093.472,214.691,427.489,176.880,18.979,152.676
C09732=1093.466,214.443,427.514,176.877,18.978,152.676
C09733=1093.460,214.193,427.538,176.875,18.976,152.677
C09734=1093.455,213.945,427.563,176.871,18.974,152.677
C09735=1093.450,213.697,427.588,176.868,18.973,152.677
C09736=1093.444,213.447,427.613,176.865,18.971,152.677
C09737=1093.439,213.199,427.637,176.862,18.969,152.677
C09738=1093.433,212.949,427.662,176.859,18.968,152.678
C09739=1093.427,212.701,427.686,176.856,18.966,152.678
C09740=1093.422,212.453,427.711,176.853,18.964,152.678
C09741=1093.416,212.204,427.736,176.850,18.963,152.678
C09742=1093.411,211.955,427.760,176.848,18.962,152.678
C09743=1093.404,211.706,427.784,176.844,18.959,152.678
C09744=1093.399,211.457,427.808,176.841,18.958,152.679
C09745=1093.393,211.209,427.832,176.838,18.956,152.679
C09746=1093.387,210.960,427.858,176.835,18.955,152.679
C09747=1093.382,210.712,427.882,176.832,18.953,152.679
C09748=1093.377,210.463,427.906,176.829,18.952,152.679
C09749=1093.371,210.214,427.931,176.827,18.950,152.680
C09750=1093.365,209.965,427.955,176.823,18.948,152.680
C09751=1093.357,209.589,427.992,176.819,18.946,152.680
C09752=1093.348,209.213,428.029,176.815,18.944,152.680
C09753=1093.340,208.837,428.066,176.810,18.942,152.681
C09754=1093.331,208.460,428.101,176.805,18.939,152.681
C09755=1093.309,207.443,428.200,176.747,18.912,152.686
C09756=1093.303,207.194,428.224,176.744,18.911,152.686
C09757=1093.297,206.945,428.248,176.740,18.911,152.687
C09758=1093.291,206.697,428.272,176.737,18.910,152.687
C09759=1093.286,206.448,428.296,176.734,18.909,152.687
C09760=1093.280,206.199,428.320,176.731,18.909,152.688
C09761=1093.274,205.950,428.344,176.728,18.908,152.688
C09762=1093.269,205.701,428.368,176.725,18.907,152.688
C09763=1093.263,205.452,428.391,176.722,18.907,152.689
C09764=1093.258,205.204,428.416,176.719,18.906,152.689
C09765=1093.252,204.955,428.439,176.716,18.905,152.690
C09766=1093.247,204.706,428.463,176.713,18.904,152.690
C09767=1093.241,204.457,428.488,176.710,18.904,152.690
C09768=1093.235,204.208,428.510,176.707,18.903,152.691
C09769=1093.230,203.960,428.535,176.704,18.902,152.691
C09770=1093.224,203.711,428.558,176.701,18.902,152.692
C09771=1093.219,203.462,428.582,176.698,18.901,152.692
C09772=1093.214,203.214,428.606,176.694,18.900,152.692
C09773=1093.208,202.965,428.629,176.691,18.899,152.693
C09774=1093.203,202.716,428.653,176.688,18.898,152.693
C09775=1093.196,202.466,428.677,176.685,18.898,152.694
C09776=1093.190,202.218,428.700,176.682,18.897,152.694
C09777=1093.185,201.969,428.724,176.679,18.897,152.695
C09778=1093.179,201.721,428.748,176.676,18.896,152.695
C09779=1093.174,201.472,428.771,176.673,18.895,152.695
C09780=1093.168,201.223,428.795,176.670,18.895,152.696
C09781=1093.162,200.974,428.818,176.667,18.894,152.696
C09782=1093.157,200.725,428.842,176.663,18.893,152.697
C09783=1093.151,200.476,428.865,176.660,18.892,152.697
C09784=1093.145,200.228,428.889,176.657,18.892,152.697
C09785=1093.140,199.979,428.913,176.654,18.891,152.698
C09786=1093.134,199.730,428.936,176.651,18.890,152.698
C09787=1093.129,199.481,428.960,176.648,18.890,152.699
C09788=1093.123,199.232,428.983,176.645,18.889,152.699
C09789=1093.117,198.983,429.007,176.642,18.889,152.700
C09790=1093.112,198.734,429.030,176.639,18.888,152.700
C09791=1093.106,198.485,429.053,176.636,18.887,152.700
C09792=1093.100,198.237,429.077,176.633,18.887,152.701
C09793=1093.095,197.988,429.100,176.630,18.886,152.701
C09794=1093.089,197.739,429.124,176.627,18.885,152.702
C09795=1093.083,197.491,429.147,176.623,18.884,152.702
C09796=1093.077,197.242,429.170,176.620,18.883,152.702
C09797=1093.072,196.992,429.193,176.617,18.883,152.703
C09798=1093.066,196.744,429.217,176.614,18.882,152.703
C09799=1093.061,196.495,429.240,176.611,18.881,152.704
C09800=1093.056,196.246,429.264,176.608,18.881,152.704
C09801=1093.050,195.997,429.287,176.605,18.880,152.704
C09802=1093.044,195.749,429.310,176.602,18.879,152.705
C09803=1093.038,195.500,429.333,176.599,18.879,152.705
C09804=1093.033,195.251,429.357,176.596,18.878,152.706
C09805=1093.027,195.002,429.380,176.593,18.877,152.706
C09806=1093.021,194.754,429.403,176.590,18.876,152.706
C09807=1093.016,194.504,429.427,176.587,18.876,152.707
C09808=1093.011,194.256,429.450,176.584,18.875,152.707
C09809=1093.005,194.007,429.473,176.581,18.874,152.707
C09810=1092.999,193.758,429.496,176.578,18.874,152.708
C09811=1092.993,193.509,429.519,176.574,18.872,152.708
C09812=1092.988,193.260,429.542,176.571,18.872,152.709
C09813=1092.982,193.011,429.566,176.568,18.871,152.709
C09814=1092.977,192.762,429.589,176.565,18.870,152.709
C09815=1092.971,192.514,429.612,176.562,18.870,152.710
C09816=1092.965,192.238,429.637,176.559,18.869,152.710
C09817=1092.959,191.961,429.663,176.556,18.868,152.711
C09818=1092.953,191.686,429.689,176.553,18.867,152.711
C09819=1092.947,191.410,429.713,176.550,18.867,152.711
C09820=1092.941,191.161,429.736,176.547,18.866,152.712
C09821=1092.936,190.912,429.760,176.544,18.865,152.712
C09822=1092.930,190.663,429.783,176.541,18.864,152.712
C09823=1092.925,190.414,429.806,176.538,18.863,152.713
C09824=1092.919,190.166,429.829,176.535,18.863,152.713
C09825=1092.913,189.917,429.852,176.532,18.862,152.714
C09826=1092.908,189.667,429.875,176.529,18.861,152.714
C09827=1092.903,189.419,429.898,176.526,18.861,152.714
C09828=1092.897,189.170,429.921,176.523,18.860,152.715
C09829=1092.892,188.921,429.944,176.519,18.858,152.715
C09830=1092.886,188.673,429.967,176.516,18.858,152.716
C09831=1092.880,188.424,429.990,176.513,18.857,152.716
C09832=1092.874,188.175,430.013,176.510,18.857,152.716
C09833=1092.869,187.926,430.036,176.507,18.855,152.717
C09834=1092.864,187.677,430.059,176.504,18.855,152.717
C09835=1092.859,187.428,430.081,176.501,18.854,152.717
C09836=1092.853,187.179,430.104,176.498,18.853,152.718
C09837=1092.847,186.930,430.127,176.496,18.852,152.718
C09838=1092.842,186.681,430.150,176.493,18.852,152.718
C09839=1092.836,186.433,430.172,176.490,18.851,152.719
C09840=1092.831,186.184,430.195,176.487,18.850,152.719
C09841=1092.825,185.935,430.218,176.484,18.849,152.720
C09842=1092.820,185.686,430.241,176.481,18.848,152.720
C09843=1092.815,185.437,430.264,176.478,18.848,152.720
C09844=1092.809,185.188,430.287,176.475,18.847,152.721
C09845=1092.803,184.939,430.308,176.472,18.846,152.721
C09846=1092.798,184.690,430.331,176.469,18.845,152.721
C09847=1092.792,184.441,430.354,176.466,18.845,152.722
C09848=1092.786,184.192,430.377,176.463,18.844,152.722
C09849=1092.781,183.943,430.399,176.460,18.843,152.723
C09850=1092.774,183.694,430.422,176.457,18.843,152.723
C09851=1092.769,183.446,430.444,176.454,18.842,152.723
C09852=1092.763,183.197,430.467,176.451,18.841,152.724
C09853=1092.758,182.948,430.489,176.449,18.840,152.724
C09854=1092.751,182.699,430.512,176.446,18.840,152.724
C09855=1092.746,182.450,430.535,176.443,18.839,152.725
C09856=1092.740,182.201,430.557,176.440,18.838,152.725
C09857=1092.735,181.952,430.580,176.437,18.838,152.726
C09858=1092.729,181.703,430.601,176.434,18.837,152.726
C09859=1092.723,181.454,430.624,176.431,18.836,152.726
C09860=1092.718,181.205,430.647,176.429,18.836,152.727
C09861=1092.712,180.956,430.669,176.426,18.835,152.727
C09862=1092.706,180.707,430.692,176.423,18.834,152.727
C09863=1092.701,180.459,430.714,176.420,18.834,152.728
C09864=1092.695,180.210,430.736,176.417,18.833,152.728
C09865=1092.689,179.960,430.758,176.414,18.832,152.729
C09866=1092.683,179.712,430.781,176.411,18.831,152.729
C09867=1092.678,179.463,430.804,176.408,18.831,152.729
C09868=1092.672,179.214,430.825,176.405,18.830,152.730
C09869=1092.666,178.965,430.848,176.402,18.829,152.730
C09870=1092.661,178.716,430.870,176.399,18.828,152.730
C09871=1092.655,178.468,430.892,176.396,18.828,152.731
C09872=1092.649,178.218,430.915,176.393,18.827,152.731
C09873=1092.644,177.969,430.937,176.390,18.826,152.731
C09874=1092.638,177.720,430.959,176.387,18.825,152.732
C09875=1092.633,177.471,430.981,176.384,18.825,152.732
C09876=1092.627,177.223,431.004,176.381,18.824,152.733
C09877=1092.621,176.973,431.026,176.379,18.823,152.733
C09878=1092.615,176.724,431.049,176.376,18.822,152.733
C09879=1092.610,176.476,431.070,176.373,18.821,152.734
C09880=1092.604,176.200,431.095,176.370,18.821,152.734
C09881=1092.597,175.923,431.119,176.367,18.820,152.734
C09882=1092.591,175.647,431.144,176.363,18.818,152.735
C09883=1092.585,175.371,431.168,176.360,18.818,152.735
C09884=1092.579,175.122,431.191,176.357,18.817,152.736
C09885=1092.574,174.873,431.213,176.354,18.816,152.736
C09886=1092.568,174.625,431.235,176.351,18.815,152.736
C09887=1092.563,174.375,431.257,176.348,18.815,152.737
C09888=1092.557,174.126,431.279,176.346,18.814,152.737
C09889=1092.551,173.878,431.301,176.343,18.814,152.737
C09890=1092.546,173.628,431.323,176.340,18.813,152.738
C09891=1092.540,173.380,431.345,176.338,18.812,152.738
C09892=1092.535,173.130,431.367,176.335,18.811,152.738
C09893=1092.528,172.881,431.389,176.332,18.810,152.739
C09894=1092.524,172.633,431.411,176.329,18.809,152.739
C09895=1092.518,172.383,431.433,176.326,18.809,152.739
C09896=1092.513,172.135,431.455,176.323,18.808,152.740
C09897=1092.506,171.886,431.477,176.320,18.807,152.740
C09898=1092.501,171.637,431.499,176.317,18.806,152.740
C09899=1092.496,171.388,431.521,176.314,18.805,152.741
C09900=1092.490,171.139,431.543,176.312,18.804,152.741
C09901=1092.485,170.890,431.565,176.309,18.803,152.741
C09902=1092.479,170.641,431.586,176.306,18.802,152.742
C09903=1092.474,170.392,431.608,176.304,18.802,152.742
C09904=1092.468,170.143,431.630,176.301,18.801,152.742
C09905=1092.462,169.894,431.653,176.298,18.800,152.743
C09906=1092.457,169.645,431.674,176.295,18.799,152.743
C09907=1092.451,169.396,431.696,176.292,18.799,152.743
C09908=1092.446,169.147,431.717,176.290,18.797,152.744
C09909=1092.440,168.898,431.740,176.287,18.797,152.744
C09910=1092.435,168.649,431.761,176.284,18.796,152.744
C09911=1092.429,168.400,431.783,176.281,18.795,152.745
C09912=1092.424,168.151,431.804,176.278,18.794,152.745
C09913=1092.418,167.902,431.827,176.275,18.793,152.745
C09914=1092.413,167.653,431.848,176.272,18.792,152.746
C09915=1092.407,167.403,431.870,176.270,18.792,152.746
C09916=1092.402,167.155,431.891,176.267,18.791,152.746
C09917=1092.396,166.905,431.914,176.265,18.790,152.747
C09918=1092.391,166.657,431.935,176.262,18.789,152.747
C09919=1092.385,166.407,431.957,176.259,18.788,152.747
C09920=1092.380,166.159,431.978,176.256,18.787,152.748
C09921=1092.374,165.910,432.000,176.253,18.786,152.748
C09922=1092.369,165.661,432.022,176.250,18.785,152.748
C09923=1092.363,165.412,432.043,176.247,18.784,152.749
C09924=1092.358,165.163,432.065,176.245,18.783,152.749
C09925=1092.352,164.914,432.086,176.242,18.783,152.749
C09926=1092.347,164.664,432.108,176.240,18.782,152.749
C09927=1092.341,164.416,432.129,176.237,18.781,152.750
C09928=1092.336,164.167,432.151,176.234,18.780,152.750
C09929=1092.330,163.918,432.173,176.231,18.779,152.750
C09930=1092.325,163.669,432.194,176.229,18.778,152.751
C09931=1092.319,163.420,432.216,176.226,18.777,152.751
C09932=1092.314,163.171,432.237,176.223,18.776,152.751
C09933=1092.309,162.922,432.258,176.220,18.775,152.752
C09934=1092.303,162.673,432.281,176.218,18.775,152.752
C09935=1092.298,162.424,432.302,176.215,18.774,152.752
C09936=1092.293,162.175,432.324,176.212,18.773,152.752
C09937=1092.287,161.925,432.345,176.210,18.772,152.753
C09938=1092.281,161.677,432.366,176.207,18.771,152.753
C09939=1092.276,161.427,432.388,176.204,18.770,152.753
C09940=1092.270,161.179,432.409,176.201,18.769,152.754
C09941=1092.265,160.930,432.430,176.198,18.768,152.754
C09942=1092.259,160.681,432.452,176.196,18.768,152.754
C09943=1092.253,160.432,432.473,176.193,18.767,152.755
C09944=1092.248,160.155,432.496,176.190,18.765,152.755
C09945=1092.241,159.878,432.520,176.187,18.765,152.755
C09946=1092.234,159.602,432.544,176.184,18.764,152.756
C09947=1092.228,159.326,432.567,176.181,18.763,152.756
C09948=1092.223,159.077,432.588,176.178,18.762,152.756
C09949=1092.217,158.827,432.609,176.175,18.761,152.757
C09950=1092.211,158.579,432.631,176.172,18.760,152.757
C09951=1092.205,158.330,432.652,176.170,18.759,152.757
C09952=1092.201,158.080,432.673,176.167,18.759,152.758
C09953=1092.195,157.832,432.695,176.165,18.758,152.758
C09954=1092.189,157.582,432.716,176.162,18.757,152.758
C09955=1092.184,157.333,432.737,176.159,18.755,152.758
C09956=1092.178,157.085,432.758,176.156,18.755,152.759
C09957=1092.172,156.835,432.779,176.153,18.754,152.759
C09958=1092.167,156.587,432.800,176.152,18.753,152.759
C09959=1092.162,156.337,432.821,176.149,18.752,152.760
C09960=1092.155,156.088,432.843,176.146,18.751,152.760
C09961=1092.150,155.839,432.863,176.143,18.750,152.760
C09962=1092.145,155.591,432.884,176.140,18.749,152.760
C09963=1092.139,155.341,432.905,176.137,18.748,152.761
C09964=1092.133,155.092,432.927,176.135,18.747,152.761
C09965=1092.128,154.843,432.947,176.133,18.747,152.761
C09966=1092.122,154.594,432.969,176.130,18.746,152.762
C09967=1092.117,154.345,432.989,176.127,18.745,152.762
C09968=1092.111,154.096,433.011,176.124,18.744,152.762
C09969=1092.105,153.847,433.032,176.121,18.743,152.763
C09970=1092.100,153.597,433.052,176.118,18.742,152.763
C09971=1092.094,153.349,433.073,176.116,18.742,152.763
C09972=1092.089,153.100,433.094,176.114,18.740,152.763
C09973=1092.083,152.851,433.116,176.111,18.739,152.764
C09974=1092.078,152.601,433.136,176.108,18.739,152.764
C09975=1092.072,152.352,433.157,176.105,18.738,152.764
C09976=1092.066,152.103,433.178,176.102,18.736,152.765
C09977=1092.061,151.854,433.199,176.101,18.736,152.765
C09978=1092.056,151.605,433.219,176.098,18.735,152.765
C09979=1092.050,151.356,433.241,176.095,18.734,152.765
C09980=1092.044,151.107,433.261,176.092,18.733,152.766
C09981=1092.038,150.858,433.282,176.089,18.732,152.766
C09982=1092.033,150.609,433.303,176.087,18.731,152.766
C09983=1092.027,150.360,433.323,176.085,18.730,152.767
C09984=1092.022,150.110,433.344,176.082,18.729,152.767
C09985=1092.016,149.862,433.366,176.079,18.728,152.767
C09986=1092.011,149.613,433.386,176.076,18.727,152.768
C09987=1092.005,149.364,433.406,176.073,18.726,152.768
C09988=1091.999,149.114,433.427,176.071,18.726,152.768
C09989=1091.993,148.866,433.448,176.069,18.724,152.768
C09990=1091.988,148.616,433.469,176.066,18.723,152.769
C09991=1091.983,148.367,433.489,176.063,18.722,152.769
C09992=1091.978,148.118,433.510,176.060,18.721,152.769
C09993=1091.971,147.869,433.530,176.058,18.721,152.769
C09994=1091.965,147.620,433.551,176.055,18.720,152.770
C09995=1091.960,147.371,433.572,176.053,18.719,152.770
C09996=1091.955,147.122,433.593,176.050,18.718,152.770
//INST
///DATE 2021/06/25 14:44
///ATTR SC,RW,RJ
////FRAME ROBOT
///GROUP1 RB1
NOP
MOVL C00000 V=800.0 PL=0
MOVL C00001 V=800.0 PL=0
MOVL C00002 V=800.0 PL=0
MOVL C00003 V=800.0 PL=0
MOVL C00004 V=800.0 PL=0
MOVL C00005 V=800.0 PL=0
MOVL C00006 V=800.0 PL=0
MOVL C00007 V=800.0 PL=0
MOVL C00008 V=800.0 PL=0
MOVL C00009 V=800.0 PL=0
MOVL C00010 V=800.0 PL=0
MOVL C00011 V=800.0 PL=0
MOVL C00012 V=800.0 PL=0
MOVL C00013 V=800.0 PL=0
MOVL C00014 V=800.0 PL=0
MOVL C00015 V=800.0 PL=0
MOVL C00016 V=800.0 PL=0
MOVL C00017 V=800.0 PL=0
MOVL C00018 V=800.0 PL=0
MOVL C00019 V=800.0 PL=0
MOVL C00020 V=800.0 PL=0
MOVL C00021 V=800.0 PL=0
MOVL C00022 V=800.0 PL=0
MOVL C00023 V=800.0 PL=0
MOVL C00024 V=800.0 PL=0
MOVL C00025 V=800.0 PL=0
MOVL C00026 V=800.0 PL=0
MOVL C00027 V=800.0 PL=0
MOVL C00028 V=800.0 PL=0
MOVL C00029 V=800.0 PL=0
MOVL C00030 V=800.0 PL=0
MOVL C00031 V=800.0 PL=0
MOVL C00032 V=800.0 PL=0
MOVL C00033 V=800.0 PL=0
MOVL C00034 V=800.0 PL=0
MOVL C00035 V=800.0 PL=0
MOVL C00036 V=800.0 PL=0
MOVL C00037 V=800.0 PL=0
MOVL C00038 V=800.0 PL=0
MOVL C00039 V=800.0 PL=0
MOVL C00040 V=800.0 PL=0
MOVL C00041 V=800.0 PL=0
MOVL C00042 V=800.0 PL=0
MOVL C00043 V=800.0 PL=0
MOVL C00044 V=800.0 PL=0
MOVL C00045 V=800.0 PL=0
MOVL C00046 V=800.0 PL=0
MOVL C00047 V=800.0 PL=0
MOVL C00048 V=800.0 PL=0
MOVL C00049 V=800.0 PL=0
MOVL C00050 V=800.0 PL=0
MOVL C00051 V=800.0 PL=0
MOVL C00052 V=800.0 PL=0
MOVL C00053 V=800.0 PL=0
MOVL C00054 V=800.0 PL=0
MOVL C00055 V=800.0 PL=0
MOVL C00056 V=800.0 PL=0
MOVL C00057 V=800.0 PL=0
MOVL C00058 V=800.0 PL=0
MOVL C00059 V=800.0 PL=0
MOVL C00060 V=800.0 PL=0
MOVL C00061 V=800.0 PL=0
MOVL C00062 V=800.0 PL=0
MOVL C00063 V=800.0 PL=0
MOVL C00064 V=800.0 PL=0
MOVL C00065 V=800.0 PL=0
MOVL C00066 V=800.0 PL=0
MOVL C00067 V=800.0 PL=0
MOVL C00068 V=800.0 PL=0
MOVL C00069 V=800.0 PL=0
MOVL C00070 V=800.0 PL=0
MOVL C00071 V=800.0 PL=0
MOVL C00072 V=800.0 PL=0
MOVL C00073 V=800.0 PL=0
MOVL C00074 V=800.0 PL=0
MOVL C00075 V=800.0 PL=0
MOVL C00076 V=800.0 PL=0
MOVL C00077 V=800.0 PL=0
MOVL C00078 V=800.0 PL=0
MOVL C00079 V=800.0 PL=0
MOVL C00080 V=800.0 PL=0
MOVL C00081 V=800.0 PL=0
MOVL C00082 V=800.0 PL=0
MOVL C00083 V=800.0 PL=0
MOVL C00084 V=800.0 PL=0
MOVL C00085 V=800.0 PL=0
MOVL C00086 V=800.0 PL=0
MOVL C00087 V=800.0 PL=0
MOVL C00088 V=800.0 PL=0
MOVL C00089 V=800.0 PL=0
MOVL C00090 V=800.0 PL=0
MOVL C00091 V=800.0 PL=0
MOVL C00092 V=800.0 PL=0
MOVL C00093 V=800.0 PL=0
MOVL C00094 V=800.0 PL=0
MOVL C00095 V=800.0 PL=0
MOVL C00096 V=800.0 PL=0
MOVL C00097 V=800.0 PL=0
MOVL C00098 V=800.0 PL=0
MOVL C00099 V=800.0 PL=0
MOVL C00100 V=800.0 PL=0
MOVL C00101 V=800.0 PL=0
MOVL C00102 V=800.0 PL=0
MOVL C00103 V=800.0 PL=0
MOVL C00104 V=800.0 PL=0
MOVL C00105 V=800.0 PL=0
MOVL C00106 V=800.0 PL=0
MOVL C00107 V=800.0 PL=0
MOVL C00108 V=800.0 PL=0
MOVL C00109 V=800.0 PL=0
MOVL C00110 V=800.0 PL=0
MOVL C00111 V=800.0 PL=0
MOVL C00112 V=800.0 PL=0
MOVL C00113 V=800.0 PL=0
MOVL C00114 V=800.0 PL=0
MOVL C00115 V=800.0 PL=0
MOVL C00116 V=800.0 PL=0
MOVL C00117 V=800.0 PL=0
MOVL C00118 V=800.0 PL=0
MOVL C00119 V=800.0 PL=0
MOVL C00120 V=800.0 PL=0
MOVL C00121 V=800.0 PL=0
MOVL C00122 V=800.0 PL=0
MOVL C00123 V=800.0 PL=0
MOVL C00124 V=800.0 PL=0
MOVL C00125 V=800.0 PL=0
MOVL C00126 V=800.0 PL=0
MOVL C00127 V=800.0 PL=0
MOVL C00128 V=800.0 PL=0
MOVL C00129 V=800.0 PL=0
MOVL C00130 V=800.0 PL=0
MOVL C00131 V=800.0 PL=0
MOVL C00132 V=800.0 PL=0
MOVL C00133 V=800.0 PL=0
MOVL C00134 V=800.0 PL=0
MOVL C00135 V=800.0 PL=0
MOVL C00136 V=800.0 PL=0
MOVL C00137 V=800.0 PL=0
MOVL C00138 V=800.0 PL=0
MOVL C00139 V=800.0 PL=0
MOVL C00140 V=800.0 PL=0
MOVL C00141 V=800.0 PL=0
MOVL C00142 V=800.0 PL=0
MOVL C00143 V=800.0 PL=0
MOVL C00144 V=800.0 PL=0
MOVL C00145 V=800.0 PL=0
MOVL C00146 V=800.0 PL=0
MOVL C00147 V=800.0 PL=0
MOVL C00148 V=800.0 PL=0
MOVL C00149 V=800.0 PL=0
MOVL C00150 V=800.0 PL=0
MOVL C00151 V=800.0 PL=0
MOVL C00152 V=800.0 PL=0
MOVL C00153 V=800.0 PL=0
MOVL C00154 V=800.0 PL=0
MOVL C00155 V=800.0 PL=0
MOVL C00156 V=800.0 PL=0
MOVL C00157 V=800.0 PL=0
MOVL C00158 V=800.0 PL=0
MOVL C00159 V=800.0 PL=0
MOVL C00160 V=800.0 PL=0
MOVL C00161 V=800.0 PL=0
MOVL C00162 V=800.0 PL=0
MOVL C00163 V=800.0 PL=0
MOVL C00164 V=800.0 PL=0
MOVL C00165 V=800.0 PL=0
MOVL C00166 V=800.0 PL=0
MOVL C00167 V=800.0 PL=0
MOVL C00168 V=800.0 PL=0
MOVL C00169 V=800.0 PL=0
MOVL C00170 V=800.0 PL=0
MOVL C00171 V=800.0 PL=0
MOVL C00172 V=800.0 PL=0
MOVL C00173 V=800.0 PL=0
MOVL C00174 V=800.0 PL=0
MOVL C00175 V=800.0 PL=0
MOVL C00176 V=800.0 PL=0
MOVL C00177 V=800.0 PL=0
MOVL C00178 V=800.0 PL=0
MOVL C00179 V=800.0 PL=0
MOVL C00180 V=800.0 PL=0
MOVL C00181 V=800.0 PL=0
MOVL C00182 V=800.0 PL=0
MOVL C00183 V=800.0 PL=0
MOVL C00184 V=800.0 PL=0
MOVL C00185 V=800.0 PL=0
MOVL C00186 V=800.0 PL=0
MOVL C00187 V=800.0 PL=0
MOVL C00188 V=800.0 PL=0
MOVL C00189 V=800.0 PL=0
MOVL C00190 V=800.0 PL=0
MOVL C00191 V=800.0 PL=0
MOVL C00192 V=800.0 PL=0
MOVL C00193 V=800.0 PL=0
MOVL C00194 V=800.0 PL=0
MOVL C00195 V=800.0 PL=0
MOVL C00196 V=800.0 PL=0
MOVL C00197 V=800.0 PL=0
MOVL C00198 V=800.0 PL=0
MOVL C00199 V=800.0 PL=0
MOVL C00200 V=800.0 PL=0
MOVL C00201 V=800.0 PL=0
MOVL C00202 V=800.0 PL=0
MOVL C00203 V=800.0 PL=0
MOVL C00204 V=800.0 PL=0
MOVL C00205 V=800.0 PL=0
MOVL C00206 V=800.0 PL=0
MOVL C00207 V=800.0 PL=0
MOVL C00208 V=800.0 PL=0
MOVL C00209 V=800.0 PL=0
MOVL C00210 V=800.0 PL=0
MOVL C00211 V=800.0 PL=0
MOVL C00212 V=800.0 PL=0
MOVL C00213 V=800.0 PL=0
MOVL C00214 V=800.0 PL=0
MOVL C00215 V=800.0 PL=0
MOVL C00216 V=800.0 PL=0
MOVL C00217 V=800.0 PL=0
MOVL C00218 V=800.0 PL=0
MOVL C00219 V=800.0 PL=0
MOVL C00220 V=800.0 PL=0
MOVL C00221 V=800.0 PL=0
MOVL C00222 V=800.0 PL=0
MOVL C00223 V=800.0 PL=0
MOVL C00224 V=800.0 PL=0
MOVL C00225 V=800.0 PL=0
MOVL C00226 V=800.0 PL=0
MOVL C00227 V=800.0 PL=0
MOVL C00228 V=800.0 PL=0
MOVL C00229 V=800.0 PL=0
MOVL C00230 V=800.0 PL=0
MOVL C00231 V=800.0 PL=0
MOVL C00232 V=800.0 PL=0
MOVL C00233 V=800.0 PL=0
MOVL C00234 V=800.0 PL=0
MOVL C00235 V=800.0 PL=0
MOVL C00236 V=800.0 PL=0
MOVL C00237 V=800.0 PL=0
MOVL C00238 V=800.0 PL=0
MOVL C00239 V=800.0 PL=0
MOVL C00240 V=800.0 PL=0
MOVL C00241 V=800.0 PL=0
MOVL C00242 V=800.0 PL=0
MOVL C00243 V=800.0 PL=0
MOVL C00244 V=800.0 PL=0
MOVL C00245 V=800.0 PL=0
MOVL C00246 V=800.0 PL=0
MOVL C00247 V=800.0 PL=0
MOVL C00248 V=800.0 PL=0
MOVL C00249 V=800.0 PL=0
MOVL C00250 V=800.0 PL=0
MOVL C00251 V=800.0 PL=0
MOVL C00252 V=800.0 PL=0
MOVL C00253 V=800.0 PL=0
MOVL C00254 V=800.0 PL=0
MOVL C00255 V=800.0 PL=0
MOVL C00256 V=800.0 PL=0
MOVL C00257 V=800.0 PL=0
MOVL C00258 V=800.0 PL=0
MOVL C00259 V=800.0 PL=0
MOVL C00260 V=800.0 PL=0
MOVL C00261 V=800.0 PL=0
MOVL C00262 V=800.0 PL=0
MOVL C00263 V=800.0 PL=0
MOVL C00264 V=800.0 PL=0
MOVL C00265 V=800.0 PL=0
MOVL C00266 V=800.0 PL=0
MOVL C00267 V=800.0 PL=0
MOVL C00268 V=800.0 PL=0
MOVL C00269 V=800.0 PL=0
MOVL C00270 V=800.0 PL=0
MOVL C00271 V=800.0 PL=0
MOVL C00272 V=800.0 PL=0
MOVL C00273 V=800.0 PL=0
MOVL C00274 V=800.0 PL=0
MOVL C00275 V=800.0 PL=0
MOVL C00276 V=800.0 PL=0
MOVL C00277 V=800.0 PL=0
MOVL C00278 V=800.0 PL=0
MOVL C00279 V=800.0 PL=0
MOVL C00280 V=800.0 PL=0
MOVL C00281 V=800.0 PL=0
MOVL C00282 V=800.0 PL=0
MOVL C00283 V=800.0 PL=0
MOVL C00284 V=800.0 PL=0
MOVL C00285 V=800.0 PL=0
MOVL C00286 V=800.0 PL=0
MOVL C00287 V=800.0 PL=0
MOVL C00288 V=800.0 PL=0
MOVL C00289 V=800.0 PL=0
MOVL C00290 V=800.0 PL=0
MOVL C00291 V=800.0 PL=0
MOVL C00292 V=800.0 PL=0
MOVL C00293 V=800.0 PL=0
MOVL C00294 V=800.0 PL=0
MOVL C00295 V=800.0 PL=0
MOVL C00296 V=800.0 PL=0
MOVL C00297 V=800.0 PL=0
MOVL C00298 V=800.0 PL=0
MOVL C00299 V=800.0 PL=0
MOVL C00300 V=800.0 PL=0
MOVL C00301 V=800.0 PL=0
MOVL C00302 V=800.0 PL=0
MOVL C00303 V=800.0 PL=0
MOVL C00304 V=800.0 PL=0
MOVL C00305 V=800.0 PL=0
MOVL C00306 V=800.0 PL=0
MOVL C00307 V=800.0 PL=0
MOVL C00308 V=800.0 PL=0
MOVL C00309 V=800.0 PL=0
MOVL C00310 V=800.0 PL=0
MOVL C00311 V=800.0 PL=0
MOVL C00312 V=800.0 PL=0
MOVL C00313 V=800.0 PL=0
MOVL C00314 V=800.0 PL=0
MOVL C00315 V=800.0 PL=0
MOVL C00316 V=800.0 PL=0
MOVL C00317 V=800.0 PL=0
MOVL C00318 V=800.0 PL=0
MOVL C00319 V=800.0 PL=0
MOVL C00320 V=800.0 PL=0
MOVL C00321 V=800.0 PL=0
MOVL C00322 V=800.0 PL=0
MOVL C00323 V=800.0 PL=0
MOVL C00324 V=800.0 PL=0
MOVL C00325 V=800.0 PL=0
MOVL C00326 V=800.0 PL=0
MOVL C00327 V=800.0 PL=0
MOVL C00328 V=800.0 PL=0
MOVL C00329 V=800.0 PL=0
MOVL C00330 V=800.0 PL=0
MOVL C00331 V=800.0 PL=0
MOVL C00332 V=800.0 PL=0
MOVL C00333 V=800.0 PL=0
MOVL C00334 V=800.0 PL=0
MOVL C00335 V=800.0 PL=0
MOVL C00336 V=800.0 PL=0
MOVL C00337 V=800.0 PL=0
MOVL C00338 V=800.0 PL=0
MOVL C00339 V=800.0 PL=0
MOVL C00340 V=800.0 PL=0
MOVL C00341 V=800.0 PL=0
MOVL C00342 V=800.0 PL=0
MOVL C00343 V=800.0 PL=0
MOVL C00344 V=800.0 PL=0
MOVL C00345 V=800.0 PL=0
MOVL C00346 V=800.0 PL=0
MOVL C00347 V=800.0 PL=0
MOVL C00348 V=800.0 PL=0
MOVL C00349 V=800.0 PL=0
MOVL C00350 V=800.0 PL=0
MOVL C00351 V=800.0 PL=0
MOVL C00352 V=800.0 PL=0
MOVL C00353 V=800.0 PL=0
MOVL C00354 V=800.0 PL=0
MOVL C00355 V=800.0 PL=0
MOVL C00356 V=800.0 PL=0
MOVL C00357 V=800.0 PL=0
MOVL C00358 V=800.0 PL=0
MOVL C00359 V=800.0 PL=0
MOVL C00360 V=800.0 PL=0
MOVL C00361 V=800.0 PL=0
MOVL C00362 V=800.0 PL=0
MOVL C00363 V=800.0 PL=0
MOVL C00364 V=800.0 PL=0
MOVL C00365 V=800.0 PL=0
MOVL C00366 V=800.0 PL=0
MOVL C00367 V=800.0 PL=0
MOVL C00368 V=800.0 PL=0
MOVL C00369 V=800.0 PL=0
MOVL C00370 V=800.0 PL=0
MOVL C00371 V=800.0 PL=0
MOVL C00372 V=800.0 PL=0
MOVL C00373 V=800.0 PL=0
MOVL C00374 V=800.0 PL=0
MOVL C00375 V=800.0 PL=0
MOVL C00376 V=800.0 PL=0
MOVL C00377 V=800.0 PL=0
MOVL C00378 V=800.0 PL=0
MOVL C00379 V=800.0 PL=0
MOVL C00380 V=800.0 PL=0
MOVL C00381 V=800.0 PL=0
MOVL C00382 V=800.0 PL=0
MOVL C00383 V=800.0 PL=0
MOVL C00384 V=800.0 PL=0
MOVL C00385 V=800.0 PL=0
MOVL C00386 V=800.0 PL=0
MOVL C00387 V=800.0 PL=0
MOVL C00388 V=800.0 PL=0
MOVL C00389 V=800.0 PL=0
MOVL C00390 V=800.0 PL=0
MOVL C00391 V=800.0 PL=0
MOVL C00392 V=800.0 PL=0
MOVL C00393 V=800.0 PL=0
MOVL C00394 V=800.0 PL=0
MOVL C00395 V=800.0 PL=0
MOVL C00396 V=800.0 PL=0
MOVL C00397 V=800.0 PL=0
MOVL C00398 V=800.0 PL=0
MOVL C00399 V=800.0 PL=0
MOVL C00400 V=800.0 PL=0
MOVL C00401 V=800.0 PL=0
MOVL C00402 V=800.0 PL=0
MOVL C00403 V=800.0 PL=0
MOVL C00404 V=800.0 PL=0
MOVL C00405 V=800.0 PL=0
MOVL C00406 V=800.0 PL=0
MOVL C00407 V=800.0 PL=0
MOVL C00408 V=800.0 PL=0
MOVL C00409 V=800.0 PL=0
MOVL C00410 V=800.0 PL=0
MOVL C00411 V=800.0 PL=0
MOVL C00412 V=800.0 PL=0
MOVL C00413 V=800.0 PL=0
MOVL C00414 V=800.0 PL=0
MOVL C00415 V=800.0 PL=0
MOVL C00416 V=800.0 PL=0
MOVL C00417 V=800.0 PL=0
MOVL C00418 V=800.0 PL=0
MOVL C00419 V=800.0 PL=0
MOVL C00420 V=800.0 PL=0
MOVL C00421 V=800.0 PL=0
MOVL C00422 V=800.0 PL=0
MOVL C00423 V=800.0 PL=0
MOVL C00424 V=800.0 PL=0
MOVL C00425 V=800.0 PL=0
MOVL C00426 V=800.0 PL=0
MOVL C00427 V=800.0 PL=0
MOVL C00428 V=800.0 PL=0
MOVL C00429 V=800.0 PL=0
MOVL C00430 V=800.0 PL=0
MOVL C00431 V=800.0 PL=0
MOVL C00432 V=800.0 PL=0
MOVL C00433 V=800.0 PL=0
MOVL C00434 V=800.0 PL=0
MOVL C00435 V=800.0 PL=0
MOVL C00436 V=800.0 PL=0
MOVL C00437 V=800.0 PL=0
MOVL C00438 V=800.0 PL=0
MOVL C00439 V=800.0 PL=0
MOVL C00440 V=800.0 PL=0
MOVL C00441 V=800.0 PL=0
MOVL C00442 V=800.0 PL=0
MOVL C00443 V=800.0 PL=0
MOVL C00444 V=800.0 PL=0
MOVL C00445 V=800.0 PL=0
MOVL C00446 V=800.0 PL=0
MOVL C00447 V=800.0 PL=0
MOVL C00448 V=800.0 PL=0
MOVL C00449 V=800.0 PL=0
MOVL C00450 V=800.0 PL=0
MOVL C00451 V=800.0 PL=0
MOVL C00452 V=800.0 PL=0
MOVL C00453 V=800.0 PL=0
MOVL C00454 V=800.0 PL=0
MOVL C00455 V=800.0 PL=0
MOVL C00456 V=800.0 PL=0
MOVL C00457 V=800.0 PL=0
MOVL C00458 V=800.0 PL=0
MOVL C00459 V=800.0 PL=0
MOVL C00460 V=800.0 PL=0
MOVL C00461 V=800.0 PL=0
MOVL C00462 V=800.0 PL=0
MOVL C00463 V=800.0 PL=0
MOVL C00464 V=800.0 PL=0
MOVL C00465 V=800.0 PL=0
MOVL C00466 V=800.0 PL=0
MOVL C00467 V=800.0 PL=0
MOVL C00468 V=800.0 PL=0
MOVL C00469 V=800.0 PL=0
MOVL C00470 V=800.0 PL=0
MOVL C00471 V=800.0 PL=0
MOVL C00472 V=800.0 PL=0
MOVL C00473 V=800.0 PL=0
MOVL C00474 V=800.0 PL=0
MOVL C00475 V=800.0 PL=0
MOVL C00476 V=800.0 PL=0
MOVL C00477 V=800.0 PL=0
MOVL C00478 V=800.0 PL=0
MOVL C00479 V=800.0 PL=0
MOVL C00480 V=800.0 PL=0
MOVL C00481 V=800.0 PL=0
MOVL C00482 V=800.0 PL=0
MOVL C00483 V=800.0 PL=0
MOVL C00484 V=800.0 PL=0
MOVL C00485 V=800.0 PL=0
MOVL C00486 V=800.0 PL=0
MOVL C00487 V=800.0 PL=0
MOVL C00488 V=800.0 PL=0
MOVL C00489 V=800.0 PL=0
MOVL C00490 V=800.0 PL=0
MOVL C00491 V=800.0 PL=0
MOVL C00492 V=800.0 PL=0
MOVL C00493 V=800.0 PL=0
MOVL C00494 V=800.0 PL=0
MOVL C00495 V=800.0 PL=0
MOVL C00496 V=800.0 PL=0
MOVL C00497 V=800.0 PL=0
MOVL C00498 V=800.0 PL=0
MOVL C00499 V=800.0 PL=0
MOVL C00500 V=800.0 PL=0
MOVL C00501 V=800.0 PL=0
MOVL C00502 V=800.0 PL=0
MOVL C00503 V=800.0 PL=0
MOVL C00504 V=800.0 PL=0
MOVL C00505 V=800.0 PL=0
MOVL C00506 V=800.0 PL=0
MOVL C00507 V=800.0 PL=0
MOVL C00508 V=800.0 PL=0
MOVL C00509 V=800.0 PL=0
MOVL C00510 V=800.0 PL=0
MOVL C00511 V=800.0 PL=0
MOVL C00512 V=800.0 PL=0
MOVL C00513 V=800.0 PL=0
MOVL C00514 V=800.0 PL=0
MOVL C00515 V=800.0 PL=0
MOVL C00516 V=800.0 PL=0
MOVL C00517 V=800.0 PL=0
MOVL C00518 V=800.0 PL=0
MOVL C00519 V=800.0 PL=0
MOVL C00520 V=800.0 PL=0
MOVL C00521 V=800.0 PL=0
MOVL C00522 V=800.0 PL=0
MOVL C00523 V=800.0 PL=0
MOVL C00524 V=800.0 PL=0
MOVL C00525 V=800.0 PL=0
MOVL C00526 V=800.0 PL=0
MOVL C00527 V=800.0 PL=0
MOVL C00528 V=800.0 PL=0
MOVL C00529 V=800.0 PL=0
MOVL C00530 V=800.0 PL=0
MOVL C00531 V=800.0 PL=0
MOVL C00532 V=800.0 PL=0
MOVL C00533 V=800.0 PL=0
MOVL C00534 V=800.0 PL=0
MOVL C00535 V=800.0 PL=0
MOVL C00536 V=800.0 PL=0
MOVL C00537 V=800.0 PL=0
MOVL C00538 V=800.0 PL=0
MOVL C00539 V=800.0 PL=0
MOVL C00540 V=800.0 PL=0
MOVL C00541 V=800.0 PL=0
MOVL C00542 V=800.0 PL=0
MOVL C00543 V=800.0 PL=0
MOVL C00544 V=800.0 PL=0
MOVL C00545 V=800.0 PL=0
MOVL C00546 V=800.0 PL=0
MOVL C00547 V=800.0 PL=0
MOVL C00548 V=800.0 PL=0
MOVL C00549 V=800.0 PL=0
MOVL C00550 V=800.0 PL=0
MOVL C00551 V=800.0 PL=0
MOVL C00552 V=800.0 PL=0
MOVL C00553 V=800.0 PL=0
MOVL C00554 V=800.0 PL=0
MOVL C00555 V=800.0 PL=0
MOVL C00556 V=800.0 PL=0
MOVL C00557 V=800.0 PL=0
MOVL C00558 V=800.0 PL=0
MOVL C00559 V=800.0 PL=0
MOVL C00560 V=800.0 PL=0
MOVL C00561 V=800.0 PL=0
MOVL C00562 V=800.0 PL=0
MOVL C00563 V=800.0 PL=0
MOVL C00564 V=800.0 PL=0
MOVL C00565 V=800.0 PL=0
MOVL C00566 V=800.0 PL=0
MOVL C00567 V=800.0 PL=0
MOVL C00568 V=800.0 PL=0
MOVL C00569 V=800.0 PL=0
MOVL C00570 V=800.0 PL=0
MOVL C00571 V=800.0 PL=0
MOVL C00572 V=800.0 PL=0
MOVL C00573 V=800.0 PL=0
MOVL C00574 V=800.0 PL=0
MOVL C00575 V=800.0 PL=0
MOVL C00576 V=800.0 PL=0
MOVL C00577 V=800.0 PL=0
MOVL C00578 V=800.0 PL=0
MOVL C00579 V=800.0 PL=0
MOVL C00580 V=800.0 PL=0
MOVL C00581 V=800.0 PL=0
MOVL C00582 V=800.0 PL=0
MOVL C00583 V=800.0 PL=0
MOVL C00584 V=800.0 PL=0
MOVL C00585 V=800.0 PL=0
MOVL C00586 V=800.0 PL=0
MOVL C00587 V=800.0 PL=0
MOVL C00588 V=800.0 PL=0
MOVL C00589 V=800.0 PL=0
MOVL C00590 V=800.0 PL=0
MOVL C00591 V=800.0 PL=0
MOVL C00592 V=800.0 PL=0
MOVL C00593 V=800.0 PL=0
MOVL C00594 V=800.0 PL=0
MOVL C00595 V=800.0 PL=0
MOVL C00596 V=800.0 PL=0
MOVL C00597 V=800.0 PL=0
MOVL C00598 V=800.0 PL=0
MOVL C00599 V=800.0 PL=0
MOVL C00600 V=800.0 PL=0
MOVL C00601 V=800.0 PL=0
MOVL C00602 V=800.0 PL=0
MOVL C00603 V=800.0 PL=0
MOVL C00604 V=800.0 PL=0
MOVL C00605 V=800.0 PL=0
MOVL C00606 V=800.0 PL=0
MOVL C00607 V=800.0 PL=0
MOVL C00608 V=800.0 PL=0
MOVL C00609 V=800.0 PL=0
MOVL C00610 V=800.0 PL=0
MOVL C00611 V=800.0 PL=0
MOVL C00612 V=800.0 PL=0
MOVL C00613 V=800.0 PL=0
MOVL C00614 V=800.0 PL=0
MOVL C00615 V=800.0 PL=0
MOVL C00616 V=800.0 PL=0
MOVL C00617 V=800.0 PL=0
MOVL C00618 V=800.0 PL=0
MOVL C00619 V=800.0 PL=0
MOVL C00620 V=800.0 PL=0
MOVL C00621 V=800.0 PL=0
MOVL C00622 V=800.0 PL=0
MOVL C00623 V=800.0 PL=0
MOVL C00624 V=800.0 PL=0
MOVL C00625 V=800.0 PL=0
MOVL C00626 V=800.0 PL=0
MOVL C00627 V=800.0 PL=0
MOVL C00628 V=800.0 PL=0
MOVL C00629 V=800.0 PL=0
MOVL C00630 V=800.0 PL=0
MOVL C00631 V=800.0 PL=0
MOVL C00632 V=800.0 PL=0
MOVL C00633 V=800.0 PL=0
MOVL C00634 V=800.0 PL=0
MOVL C00635 V=800.0 PL=0
MOVL C00636 V=800.0 PL=0
MOVL C00637 V=800.0 PL=0
MOVL C00638 V=800.0 PL=0
MOVL C00639 V=800.0 PL=0
MOVL C00640 V=800.0 PL=0
MOVL C00641 V=800.0 PL=0
MOVL C00642 V=800.0 PL=0
MOVL C00643 V=800.0 PL=0
MOVL C00644 V=800.0 PL=0
MOVL C00645 V=800.0 PL=0
MOVL C00646 V=800.0 PL=0
MOVL C00647 V=800.0 PL=0
MOVL C00648 V=800.0 PL=0
MOVL C00649 V=800.0 PL=0
MOVL C00650 V=800.0 PL=0
MOVL C00651 V=800.0 PL=0
MOVL C00652 V=800.0 PL=0
MOVL C00653 V=800.0 PL=0
MOVL C00654 V=800.0 PL=0
MOVL C00655 V=800.0 PL=0
MOVL C00656 V=800.0 PL=0
MOVL C00657 V=800.0 PL=0
MOVL C00658 V=800.0 PL=0
MOVL C00659 V=800.0 PL=0
MOVL C00660 V=800.0 PL=0
MOVL C00661 V=800.0 PL=0
MOVL C00662 V=800.0 PL=0
MOVL C00663 V=800.0 PL=0
MOVL C00664 V=800.0 PL=0
MOVL C00665 V=800.0 PL=0
MOVL C00666 V=800.0 PL=0
MOVL C00667 V=800.0 PL=0
MOVL C00668 V=800.0 PL=0
MOVL C00669 V=800.0 PL=0
MOVL C00670 V=800.0 PL=0
MOVL C00671 V=800.0 PL=0
MOVL C00672 V=800.0 PL=0
MOVL C00673 V=800.0 PL=0
MOVL C00674 V=800.0 PL=0
MOVL C00675 V=800.0 PL=0
MOVL C00676 V=800.0 PL=0
MOVL C00677 V=800.0 PL=0
MOVL C00678 V=800.0 PL=0
MOVL C00679 V=800.0 PL=0
MOVL C00680 V=800.0 PL=0
MOVL C00681 V=800.0 PL=0
MOVL C00682 V=800.0 PL=0
MOVL C00683 V=800.0 PL=0
MOVL C00684 V=800.0 PL=0
MOVL C00685 V=800.0 PL=0
MOVL C00686 V=800.0 PL=0
MOVL C00687 V=800.0 PL=0
MOVL C00688 V=800.0 PL=0
MOVL C00689 V=800.0 PL=0
MOVL C00690 V=800.0 PL=0
MOVL C00691 V=800.0 PL=0
MOVL C00692 V=800.0 PL=0
MOVL C00693 V=800.0 PL=0
MOVL C00694 V=800.0 PL=0
MOVL C00695 V=800.0 PL=0
MOVL C00696 V=800.0 PL=0
MOVL C00697 V=800.0 PL=0
MOVL C00698 V=800.0 PL=0
MOVL C00699 V=800.0 PL=0
MOVL C00700 V=800.0 PL=0
MOVL C00701 V=800.0 PL=0
MOVL C00702 V=800.0 PL=0
MOVL C00703 V=800.0 PL=0
MOVL C00704 V=800.0 PL=0
MOVL C00705 V=800.0 PL=0
MOVL C00706 V=800.0 PL=0
MOVL C00707 V=800.0 PL=0
MOVL C00708 V=800.0 PL=0
MOVL C00709 V=800.0 PL=0
MOVL C00710 V=800.0 PL=0
MOVL C00711 V=800.0 PL=0
MOVL C00712 V=800.0 PL=0
MOVL C00713 V=800.0 PL=0
MOVL C00714 V=800.0 PL=0
MOVL C00715 V=800.0 PL=0
MOVL C00716 V=800.0 PL=0
MOVL C00717 V=800.0 PL=0
MOVL C00718 V=800.0 PL=0
MOVL C00719 V=800.0 PL=0
MOVL C00720 V=800.0 PL=0
MOVL C00721 V=800.0 PL=0
MOVL C00722 V=800.0 PL=0
MOVL C00723 V=800.0 PL=0
MOVL C00724 V=800.0 PL=0
MOVL C00725 V=800.0 PL=0
MOVL C00726 V=800.0 PL=0
MOVL C00727 V=800.0 PL=0
MOVL C00728 V=800.0 PL=0
MOVL C00729 V=800.0 PL=0
MOVL C00730 V=800.0 PL=0
MOVL C00731 V=800.0 PL=0
MOVL C00732 V=800.0 PL=0
MOVL C00733 V=800.0 PL=0
MOVL C00734 V=800.0 PL=0
MOVL C00735 V=800.0 PL=0
MOVL C00736 V=800.0 PL=0
MOVL C00737 V=800.0 PL=0
MOVL C00738 V=800.0 PL=0
MOVL C00739 V=800.0 PL=0
MOVL C00740 V=800.0 PL=0
MOVL C00741 V=800.0 PL=0
MOVL C00742 V=800.0 PL=0
MOVL C00743 V=800.0 PL=0
MOVL C00744 V=800.0 PL=0
MOVL C00745 V=800.0 PL=0
MOVL C00746 V=800.0 PL=0
MOVL C00747 V=800.0 PL=0
MOVL C00748 V=800.0 PL=0
MOVL C00749 V=800.0 PL=0
MOVL C00750 V=800.0 PL=0
MOVL C00751 V=800.0 PL=0
MOVL C00752 V=800.0 PL=0
MOVL C00753 V=800.0 PL=0
MOVL C00754 V=800.0 PL=0
MOVL C00755 V=800.0 PL=0
MOVL C00756 V=800.0 PL=0
MOVL C00757 V=800.0 PL=0
MOVL C00758 V=800.0 PL=0
MOVL C00759 V=800.0 PL=0
MOVL C00760 V=800.0 PL=0
MOVL C00761 V=800.0 PL=0
MOVL C00762 V=800.0 PL=0
MOVL C00763 V=800.0 PL=0
MOVL C00764 V=800.0 PL=0
MOVL C00765 V=800.0 PL=0
MOVL C00766 V=800.0 PL=0
MOVL C00767 V=800.0 PL=0
MOVL C00768 V=800.0 PL=0
MOVL C00769 V=800.0 PL=0
MOVL C00770 V=800.0 PL=0
MOVL C00771 V=800.0 PL=0
MOVL C00772 V=800.0 PL=0
MOVL C00773 V=800.0 PL=0
MOVL C00774 V=800.0 PL=0
MOVL C00775 V=800.0 PL=0
MOVL C00776 V=800.0 PL=0
MOVL C00777 V=800.0 PL=0
MOVL C00778 V=800.0 PL=0
MOVL C00779 V=800.0 PL=0
MOVL C00780 V=800.0 PL=0
MOVL C00781 V=800.0 PL=0
MOVL C00782 V=800.0 PL=0
MOVL C00783 V=800.0 PL=0
MOVL C00784 V=800.0 PL=0
MOVL C00785 V=800.0 PL=0
MOVL C00786 V=800.0 PL=0
MOVL C00787 V=800.0 PL=0
MOVL C00788 V=800.0 PL=0
MOVL C00789 V=800.0 PL=0
MOVL C00790 V=800.0 PL=0
MOVL C00791 V=800.0 PL=0
MOVL C00792 V=800.0 PL=0
MOVL C00793 V=800.0 PL=0
MOVL C00794 V=800.0 PL=0
MOVL C00795 V=800.0 PL=0
MOVL C00796 V=800.0 PL=0
MOVL C00797 V=800.0 PL=0
MOVL C00798 V=800.0 PL=0
MOVL C00799 V=800.0 PL=0
MOVL C00800 V=800.0 PL=0
MOVL C00801 V=800.0 PL=0
MOVL C00802 V=800.0 PL=0
MOVL C00803 V=800.0 PL=0
MOVL C00804 V=800.0 PL=0
MOVL C00805 V=800.0 PL=0
MOVL C00806 V=800.0 PL=0
MOVL C00807 V=800.0 PL=0
MOVL C00808 V=800.0 PL=0
MOVL C00809 V=800.0 PL=0
MOVL C00810 V=800.0 PL=0
MOVL C00811 V=800.0 PL=0
MOVL C00812 V=800.0 PL=0
MOVL C00813 V=800.0 PL=0
MOVL C00814 V=800.0 PL=0
MOVL C00815 V=800.0 PL=0
MOVL C00816 V=800.0 PL=0
MOVL C00817 V=800.0 PL=0
MOVL C00818 V=800.0 PL=0
MOVL C00819 V=800.0 PL=0
MOVL C00820 V=800.0 PL=0
MOVL C00821 V=800.0 PL=0
MOVL C00822 V=800.0 PL=0
MOVL C00823 V=800.0 PL=0
MOVL C00824 V=800.0 PL=0
MOVL C00825 V=800.0 PL=0
MOVL C00826 V=800.0 PL=0
MOVL C00827 V=800.0 PL=0
MOVL C00828 V=800.0 PL=0
MOVL C00829 V=800.0 PL=0
MOVL C00830 V=800.0 PL=0
MOVL C00831 V=800.0 PL=0
MOVL C00832 V=800.0 PL=0
MOVL C00833 V=800.0 PL=0
MOVL C00834 V=800.0 PL=0
MOVL C00835 V=800.0 PL=0
MOVL C00836 V=800.0 PL=0
MOVL C00837 V=800.0 PL=0
MOVL C00838 V=800.0 PL=0
MOVL C00839 V=800.0 PL=0
MOVL C00840 V=800.0 PL=0
MOVL C00841 V=800.0 PL=0
MOVL C00842 V=800.0 PL=0
MOVL C00843 V=800.0 PL=0
MOVL C00844 V=800.0 PL=0
MOVL C00845 V=800.0 PL=0
MOVL C00846 V=800.0 PL=0
MOVL C00847 V=800.0 PL=0
MOVL C00848 V=800.0 PL=0
MOVL C00849 V=800.0 PL=0
MOVL C00850 V=800.0 PL=0
MOVL C00851 V=800.0 PL=0
MOVL C00852 V=800.0 PL=0
MOVL C00853 V=800.0 PL=0
MOVL C00854 V=800.0 PL=0
MOVL C00855 V=800.0 PL=0
MOVL C00856 V=800.0 PL=0
MOVL C00857 V=800.0 PL=0
MOVL C00858 V=800.0 PL=0
MOVL C00859 V=800.0 PL=0
MOVL C00860 V=800.0 PL=0
MOVL C00861 V=800.0 PL=0
MOVL C00862 V=800.0 PL=0
MOVL C00863 V=800.0 PL=0
MOVL C00864 V=800.0 PL=0
MOVL C00865 V=800.0 PL=0
MOVL C00866 V=800.0 PL=0
MOVL C00867 V=800.0 PL=0
MOVL C00868 V=800.0 PL=0
MOVL C00869 V=800.0 PL=0
MOVL C00870 V=800.0 PL=0
MOVL C00871 V=800.0 PL=0
MOVL C00872 V=800.0 PL=0
MOVL C00873 V=800.0 PL=0
MOVL C00874 V=800.0 PL=0
MOVL C00875 V=800.0 PL=0
MOVL C00876 V=800.0 PL=0
MOVL C00877 V=800.0 PL=0
MOVL C00878 V=800.0 PL=0
MOVL C00879 V=800.0 PL=0
MOVL C00880 V=800.0 PL=0
MOVL C00881 V=800.0 PL=0
MOVL C00882 V=800.0 PL=0
MOVL C00883 V=800.0 PL=0
MOVL C00884 V=800.0 PL=0
MOVL C00885 V=800.0 PL=0
MOVL C00886 V=800.0 PL=0
MOVL C00887 V=800.0 PL=0
MOVL C00888 V=800.0 PL=0
MOVL C00889 V=800.0 PL=0
MOVL C00890 V=800.0 PL=0
MOVL C00891 V=800.0 PL=0
MOVL C00892 V=800.0 PL=0
MOVL C00893 V=800.0 PL=0
MOVL C00894 V=800.0 PL=0
MOVL C00895 V=800.0 PL=0
MOVL C00896 V=800.0 PL=0
MOVL C00897 V=800.0 PL=0
MOVL C00898 V=800.0 PL=0
MOVL C00899 V=800.0 PL=0
MOVL C00900 V=800.0 PL=0
MOVL C00901 V=800.0 PL=0
MOVL C00902 V=800.0 PL=0
MOVL C00903 V=800.0 PL=0
MOVL C00904 V=800.0 PL=0
MOVL C00905 V=800.0 PL=0
MOVL C00906 V=800.0 PL=0
MOVL C00907 V=800.0 PL=0
MOVL C00908 V=800.0 PL=0
MOVL C00909 V=800.0 PL=0
MOVL C00910 V=800.0 PL=0
MOVL C00911 V=800.0 PL=0
MOVL C00912 V=800.0 PL=0
MOVL C00913 V=800.0 PL=0
MOVL C00914 V=800.0 PL=0
MOVL C00915 V=800.0 PL=0
MOVL C00916 V=800.0 PL=0
MOVL C00917 V=800.0 PL=0
MOVL C00918 V=800.0 PL=0
MOVL C00919 V=800.0 PL=0
MOVL C00920 V=800.0 PL=0
MOVL C00921 V=800.0 PL=0
MOVL C00922 V=800.0 PL=0
MOVL C00923 V=800.0 PL=0
MOVL C00924 V=800.0 PL=0
MOVL C00925 V=800.0 PL=0
MOVL C00926 V=800.0 PL=0
MOVL C00927 V=800.0 PL=0
MOVL C00928 V=800.0 PL=0
MOVL C00929 V=800.0 PL=0
MOVL C00930 V=800.0 PL=0
MOVL C00931 V=800.0 PL=0
MOVL C00932 V=800.0 PL=0
MOVL C00933 V=800.0 PL=0
MOVL C00934 V=800.0 PL=0
MOVL C00935 V=800.0 PL=0
MOVL C00936 V=800.0 PL=0
MOVL C00937 V=800.0 PL=0
MOVL C00938 V=800.0 PL=0
MOVL C00939 V=800.0 PL=0
MOVL C00940 V=800.0 PL=0
MOVL C00941 V=800.0 PL=0
MOVL C00942 V=800.0 PL=0
MOVL C00943 V=800.0 PL=0
MOVL C00944 V=800.0 PL=0
MOVL C00945 V=800.0 PL=0
MOVL C00946 V=800.0 PL=0
MOVL C00947 V=800.0 PL=0
MOVL C00948 V=800.0 PL=0
MOVL C00949 V=800.0 PL=0
MOVL C00950 V=800.0 PL=0
MOVL C00951 V=800.0 PL=0
MOVL C00952 V=800.0 PL=0
MOVL C00953 V=800.0 PL=0
MOVL C00954 V=800.0 PL=0
MOVL C00955 V=800.0 PL=0
MOVL C00956 V=800.0 PL=0
MOVL C00957 V=800.0 PL=0
MOVL C00958 V=800.0 PL=0
MOVL C00959 V=800.0 PL=0
MOVL C00960 V=800.0 PL=0
MOVL C00961 V=800.0 PL=0
MOVL C00962 V=800.0 PL=0
MOVL C00963 V=800.0 PL=0
MOVL C00964 V=800.0 PL=0
MOVL C00965 V=800.0 PL=0
MOVL C00966 V=800.0 PL=0
MOVL C00967 V=800.0 PL=0
MOVL C00968 V=800.0 PL=0
MOVL C00969 V=800.0 PL=0
MOVL C00970 V=800.0 PL=0
MOVL C00971 V=800.0 PL=0
MOVL C00972 V=800.0 PL=0
MOVL C00973 V=800.0 PL=0
MOVL C00974 V=800.0 PL=0
MOVL C00975 V=800.0 PL=0
MOVL C00976 V=800.0 PL=0
MOVL C00977 V=800.0 PL=0
MOVL C00978 V=800.0 PL=0
MOVL C00979 V=800.0 PL=0
MOVL C00980 V=800.0 PL=0
MOVL C00981 V=800.0 PL=0
MOVL C00982 V=800.0 PL=0
MOVL C00983 V=800.0 PL=0
MOVL C00984 V=800.0 PL=0
MOVL C00985 V=800.0 PL=0
MOVL C00986 V=800.0 PL=0
MOVL C00987 V=800.0 PL=0
MOVL C00988 V=800.0 PL=0
MOVL C00989 V=800.0 PL=0
MOVL C00990 V=800.0 PL=0
MOVL C00991 V=800.0 PL=0
MOVL C00992 V=800.0 PL=0
MOVL C00993 V=800.0 PL=0
MOVL C00994 V=800.0 PL=0
MOVL C00995 V=800.0 PL=0
MOVL C00996 V=800.0 PL=0
MOVL C00997 V=800.0 PL=0
MOVL C00998 V=800.0 PL=0
MOVL C00999 V=800.0 PL=0
MOVL C01000 V=800.0 PL=0
MOVL C01001 V=800.0 PL=0
MOVL C01002 V=800.0 PL=0
MOVL C01003 V=800.0 PL=0
MOVL C01004 V=800.0 PL=0
MOVL C01005 V=800.0 PL=0
MOVL C01006 V=800.0 PL=0
MOVL C01007 V=800.0 PL=0
MOVL C01008 V=800.0 PL=0
MOVL C01009 V=800.0 PL=0
MOVL C01010 V=800.0 PL=0
MOVL C01011 V=800.0 PL=0
MOVL C01012 V=800.0 PL=0
MOVL C01013 V=800.0 PL=0
MOVL C01014 V=800.0 PL=0
MOVL C01015 V=800.0 PL=0
MOVL C01016 V=800.0 PL=0
MOVL C01017 V=800.0 PL=0
MOVL C01018 V=800.0 PL=0
MOVL C01019 V=800.0 PL=0
MOVL C01020 V=800.0 PL=0
MOVL C01021 V=800.0 PL=0
MOVL C01022 V=800.0 PL=0
MOVL C01023 V=800.0 PL=0
MOVL C01024 V=800.0 PL=0
MOVL C01025 V=800.0 PL=0
MOVL C01026 V=800.0 PL=0
MOVL C01027 V=800.0 PL=0
MOVL C01028 V=800.0 PL=0
MOVL C01029 V=800.0 PL=0
MOVL C01030 V=800.0 PL=0
MOVL C01031 V=800.0 PL=0
MOVL C01032 V=800.0 PL=0
MOVL C01033 V=800.0 PL=0
MOVL C01034 V=800.0 PL=0
MOVL C01035 V=800.0 PL=0
MOVL C01036 V=800.0 PL=0
MOVL C01037 V=800.0 PL=0
MOVL C01038 V=800.0 PL=0
MOVL C01039 V=800.0 PL=0
MOVL C01040 V=800.0 PL=0
MOVL C01041 V=800.0 PL=0
MOVL C01042 V=800.0 PL=0
MOVL C01043 V=800.0 PL=0
MOVL C01044 V=800.0 PL=0
MOVL C01045 V=800.0 PL=0
MOVL C01046 V=800.0 PL=0
MOVL C01047 V=800.0 PL=0
MOVL C01048 V=800.0 PL=0
MOVL C01049 V=800.0 PL=0
MOVL C01050 V=800.0 PL=0
MOVL C01051 V=800.0 PL=0
MOVL C01052 V=800.0 PL=0
MOVL C01053 V=800.0 PL=0
MOVL C01054 V=800.0 PL=0
MOVL C01055 V=800.0 PL=0
MOVL C01056 V=800.0 PL=0
MOVL C01057 V=800.0 PL=0
MOVL C01058 V=800.0 PL=0
MOVL C01059 V=800.0 PL=0
MOVL C01060 V=800.0 PL=0
MOVL C01061 V=800.0 PL=0
MOVL C01062 V=800.0 PL=0
MOVL C01063 V=800.0 PL=0
MOVL C01064 V=800.0 PL=0
MOVL C01065 V=800.0 PL=0
MOVL C01066 V=800.0 PL=0
MOVL C01067 V=800.0 PL=0
MOVL C01068 V=800.0 PL=0
MOVL C01069 V=800.0 PL=0
MOVL C01070 V=800.0 PL=0
MOVL C01071 V=800.0 PL=0
MOVL C01072 V=800.0 PL=0
MOVL C01073 V=800.0 PL=0
MOVL C01074 V=800.0 PL=0
MOVL C01075 V=800.0 PL=0
MOVL C01076 V=800.0 PL=0
MOVL C01077 V=800.0 PL=0
MOVL C01078 V=800.0 PL=0
MOVL C01079 V=800.0 PL=0
MOVL C01080 V=800.0 PL=0
MOVL C01081 V=800.0 PL=0
MOVL C01082 V=800.0 PL=0
MOVL C01083 V=800.0 PL=0
MOVL C01084 V=800.0 PL=0
MOVL C01085 V=800.0 PL=0
MOVL C01086 V=800.0 PL=0
MOVL C01087 V=800.0 PL=0
MOVL C01088 V=800.0 PL=0
MOVL C01089 V=800.0 PL=0
MOVL C01090 V=800.0 PL=0
MOVL C01091 V=800.0 PL=0
MOVL C01092 V=800.0 PL=0
MOVL C01093 V=800.0 PL=0
MOVL C01094 V=800.0 PL=0
MOVL C01095 V=800.0 PL=0
MOVL C01096 V=800.0 PL=0
MOVL C01097 V=800.0 PL=0
MOVL C01098 V=800.0 PL=0
MOVL C01099 V=800.0 PL=0
MOVL C01100 V=800.0 PL=0
MOVL C01101 V=800.0 PL=0
MOVL C01102 V=800.0 PL=0
MOVL C01103 V=800.0 PL=0
MOVL C01104 V=800.0 PL=0
MOVL C01105 V=800.0 PL=0
MOVL C01106 V=800.0 PL=0
MOVL C01107 V=800.0 PL=0
MOVL C01108 V=800.0 PL=0
MOVL C01109 V=800.0 PL=0
MOVL C01110 V=800.0 PL=0
MOVL C01111 V=800.0 PL=0
MOVL C01112 V=800.0 PL=0
MOVL C01113 V=800.0 PL=0
MOVL C01114 V=800.0 PL=0
MOVL C01115 V=800.0 PL=0
MOVL C01116 V=800.0 PL=0
MOVL C01117 V=800.0 PL=0
MOVL C01118 V=800.0 PL=0
MOVL C01119 V=800.0 PL=0
MOVL C01120 V=800.0 PL=0
MOVL C01121 V=800.0 PL=0
MOVL C01122 V=800.0 PL=0
MOVL C01123 V=800.0 PL=0
MOVL C01124 V=800.0 PL=0
MOVL C01125 V=800.0 PL=0
MOVL C01126 V=800.0 PL=0
MOVL C01127 V=800.0 PL=0
MOVL C01128 V=800.0 PL=0
MOVL C01129 V=800.0 PL=0
MOVL C01130 V=800.0 PL=0
MOVL C01131 V=800.0 PL=0
MOVL C01132 V=800.0 PL=0
MOVL C01133 V=800.0 PL=0
MOVL C01134 V=800.0 PL=0
MOVL C01135 V=800.0 PL=0
MOVL C01136 V=800.0 PL=0
MOVL C01137 V=800.0 PL=0
MOVL C01138 V=800.0 PL=0
MOVL C01139 V=800.0 PL=0
MOVL C01140 V=800.0 PL=0
MOVL C01141 V=800.0 PL=0
MOVL C01142 V=800.0 PL=0
MOVL C01143 V=800.0 PL=0
MOVL C01144 V=800.0 PL=0
MOVL C01145 V=800.0 PL=0
MOVL C01146 V=800.0 PL=0
MOVL C01147 V=800.0 PL=0
MOVL C01148 V=800.0 PL=0
MOVL C01149 V=800.0 PL=0
MOVL C01150 V=800.0 PL=0
MOVL C01151 V=800.0 PL=0
MOVL C01152 V=800.0 PL=0
MOVL C01153 V=800.0 PL=0
MOVL C01154 V=800.0 PL=0
MOVL C01155 V=800.0 PL=0
MOVL C01156 V=800.0 PL=0
MOVL C01157 V=800.0 PL=0
MOVL C01158 V=800.0 PL=0
MOVL C01159 V=800.0 PL=0
MOVL C01160 V=800.0 PL=0
MOVL C01161 V=800.0 PL=0
MOVL C01162 V=800.0 PL=0
MOVL C01163 V=800.0 PL=0
MOVL C01164 V=800.0 PL=0
MOVL C01165 V=800.0 PL=0
MOVL C01166 V=800.0 PL=0
MOVL C01167 V=800.0 PL=0
MOVL C01168 V=800.0 PL=0
MOVL C01169 V=800.0 PL=0
MOVL C01170 V=800.0 PL=0
MOVL C01171 V=800.0 PL=0
MOVL C01172 V=800.0 PL=0
MOVL C01173 V=800.0 PL=0
MOVL C01174 V=800.0 PL=0
MOVL C01175 V=800.0 PL=0
MOVL C01176 V=800.0 PL=0
MOVL C01177 V=800.0 PL=0
MOVL C01178 V=800.0 PL=0
MOVL C01179 V=800.0 PL=0
MOVL C01180 V=800.0 PL=0
MOVL C01181 V=800.0 PL=0
MOVL C01182 V=800.0 PL=0
MOVL C01183 V=800.0 PL=0
MOVL C01184 V=800.0 PL=0
MOVL C01185 V=800.0 PL=0
MOVL C01186 V=800.0 PL=0
MOVL C01187 V=800.0 PL=0
MOVL C01188 V=800.0 PL=0
MOVL C01189 V=800.0 PL=0
MOVL C01190 V=800.0 PL=0
MOVL C01191 V=800.0 PL=0
MOVL C01192 V=800.0 PL=0
MOVL C01193 V=800.0 PL=0
MOVL C01194 V=800.0 PL=0
MOVL C01195 V=800.0 PL=0
MOVL C01196 V=800.0 PL=0
MOVL C01197 V=800.0 PL=0
MOVL C01198 V=800.0 PL=0
MOVL C01199 V=800.0 PL=0
MOVL C01200 V=800.0 PL=0
MOVL C01201 V=800.0 PL=0
MOVL C01202 V=800.0 PL=0
MOVL C01203 V=800.0 PL=0
MOVL C01204 V=800.0 PL=0
MOVL C01205 V=800.0 PL=0
MOVL C01206 V=800.0 PL=0
MOVL C01207 V=800.0 PL=0
MOVL C01208 V=800.0 PL=0
MOVL C01209 V=800.0 PL=0
MOVL C01210 V=800.0 PL=0
MOVL C01211 V=800.0 PL=0
MOVL C01212 V=800.0 PL=0
MOVL C01213 V=800.0 PL=0
MOVL C01214 V=800.0 PL=0
MOVL C01215 V=800.0 PL=0
MOVL C01216 V=800.0 PL=0
MOVL C01217 V=800.0 PL=0
MOVL C01218 V=800.0 PL=0
MOVL C01219 V=800.0 PL=0
MOVL C01220 V=800.0 PL=0
MOVL C01221 V=800.0 PL=0
MOVL C01222 V=800.0 PL=0
MOVL C01223 V=800.0 PL=0
MOVL C01224 V=800.0 PL=0
MOVL C01225 V=800.0 PL=0
MOVL C01226 V=800.0 PL=0
MOVL C01227 V=800.0 PL=0
MOVL C01228 V=800.0 PL=0
MOVL C01229 V=800.0 PL=0
MOVL C01230 V=800.0 PL=0
MOVL C01231 V=800.0 PL=0
MOVL C01232 V=800.0 PL=0
MOVL C01233 V=800.0 PL=0
MOVL C01234 V=800.0 PL=0
MOVL C01235 V=800.0 PL=0
MOVL C01236 V=800.0 PL=0
MOVL C01237 V=800.0 PL=0
MOVL C01238 V=800.0 PL=0
MOVL C01239 V=800.0 PL=0
MOVL C01240 V=800.0 PL=0
MOVL C01241 V=800.0 PL=0
MOVL C01242 V=800.0 PL=0
MOVL C01243 V=800.0 PL=0
MOVL C01244 V=800.0 PL=0
MOVL C01245 V=800.0 PL=0
MOVL C01246 V=800.0 PL=0
MOVL C01247 V=800.0 PL=0
MOVL C01248 V=800.0 PL=0
MOVL C01249 V=800.0 PL=0
MOVL C01250 V=800.0 PL=0
MOVL C01251 V=800.0 PL=0
MOVL C01252 V=800.0 PL=0
MOVL C01253 V=800.0 PL=0
MOVL C01254 V=800.0 PL=0
MOVL C01255 V=800.0 PL=0
MOVL C01256 V=800.0 PL=0
MOVL C01257 V=800.0 PL=0
MOVL C01258 V=800.0 PL=0
MOVL C01259 V=800.0 PL=0
MOVL C01260 V=800.0 PL=0
MOVL C01261 V=800.0 PL=0
MOVL C01262 V=800.0 PL=0
MOVL C01263 V=800.0 PL=0
MOVL C01264 V=800.0 PL=0
MOVL C01265 V=800.0 PL=0
MOVL C01266 V=800.0 PL=0
MOVL C01267 V=800.0 PL=0
MOVL C01268 V=800.0 PL=0
MOVL C01269 V=800.0 PL=0
MOVL C01270 V=800.0 PL=0
MOVL C01271 V=800.0 PL=0
MOVL C01272 V=800.0 PL=0
MOVL C01273 V=800.0 PL=0
MOVL C01274 V=800.0 PL=0
MOVL C01275 V=800.0 PL=0
MOVL C01276 V=800.0 PL=0
MOVL C01277 V=800.0 PL=0
MOVL C01278 V=800.0 PL=0
MOVL C01279 V=800.0 PL=0
MOVL C01280 V=800.0 PL=0
MOVL C01281 V=800.0 PL=0
MOVL C01282 V=800.0 PL=0
MOVL C01283 V=800.0 PL=0
MOVL C01284 V=800.0 PL=0
MOVL C01285 V=800.0 PL=0
MOVL C01286 V=800.0 PL=0
MOVL C01287 V=800.0 PL=0
MOVL C01288 V=800.0 PL=0
MOVL C01289 V=800.0 PL=0
MOVL C01290 V=800.0 PL=0
MOVL C01291 V=800.0 PL=0
MOVL C01292 V=800.0 PL=0
MOVL C01293 V=800.0 PL=0
MOVL C01294 V=800.0 PL=0
MOVL C01295 V=800.0 PL=0
MOVL C01296 V=800.0 PL=0
MOVL C01297 V=800.0 PL=0
MOVL C01298 V=800.0 PL=0
MOVL C01299 V=800.0 PL=0
MOVL C01300 V=800.0 PL=0
MOVL C01301 V=800.0 PL=0
MOVL C01302 V=800.0 PL=0
MOVL C01303 V=800.0 PL=0
MOVL C01304 V=800.0 PL=0
MOVL C01305 V=800.0 PL=0
MOVL C01306 V=800.0 PL=0
MOVL C01307 V=800.0 PL=0
MOVL C01308 V=800.0 PL=0
MOVL C01309 V=800.0 PL=0
MOVL C01310 V=800.0 PL=0
MOVL C01311 V=800.0 PL=0
MOVL C01312 V=800.0 PL=0
MOVL C01313 V=800.0 PL=0
MOVL C01314 V=800.0 PL=0
MOVL C01315 V=800.0 PL=0
MOVL C01316 V=800.0 PL=0
MOVL C01317 V=800.0 PL=0
MOVL C01318 V=800.0 PL=0
MOVL C01319 V=800.0 PL=0
MOVL C01320 V=800.0 PL=0
MOVL C01321 V=800.0 PL=0
MOVL C01322 V=800.0 PL=0
MOVL C01323 V=800.0 PL=0
MOVL C01324 V=800.0 PL=0
MOVL C01325 V=800.0 PL=0
MOVL C01326 V=800.0 PL=0
MOVL C01327 V=800.0 PL=0
MOVL C01328 V=800.0 PL=0
MOVL C01329 V=800.0 PL=0
MOVL C01330 V=800.0 PL=0
MOVL C01331 V=800.0 PL=0
MOVL C01332 V=800.0 PL=0
MOVL C01333 V=800.0 PL=0
MOVL C01334 V=800.0 PL=0
MOVL C01335 V=800.0 PL=0
MOVL C01336 V=800.0 PL=0
MOVL C01337 V=800.0 PL=0
MOVL C01338 V=800.0 PL=0
MOVL C01339 V=800.0 PL=0
MOVL C01340 V=800.0 PL=0
MOVL C01341 V=800.0 PL=0
MOVL C01342 V=800.0 PL=0
MOVL C01343 V=800.0 PL=0
MOVL C01344 V=800.0 PL=0
MOVL C01345 V=800.0 PL=0
MOVL C01346 V=800.0 PL=0
MOVL C01347 V=800.0 PL=0
MOVL C01348 V=800.0 PL=0
MOVL C01349 V=800.0 PL=0
MOVL C01350 V=800.0 PL=0
MOVL C01351 V=800.0 PL=0
MOVL C01352 V=800.0 PL=0
MOVL C01353 V=800.0 PL=0
MOVL C01354 V=800.0 PL=0
MOVL C01355 V=800.0 PL=0
MOVL C01356 V=800.0 PL=0
MOVL C01357 V=800.0 PL=0
MOVL C01358 V=800.0 PL=0
MOVL C01359 V=800.0 PL=0
MOVL C01360 V=800.0 PL=0
MOVL C01361 V=800.0 PL=0
MOVL C01362 V=800.0 PL=0
MOVL C01363 V=800.0 PL=0
MOVL C01364 V=800.0 PL=0
MOVL C01365 V=800.0 PL=0
MOVL C01366 V=800.0 PL=0
MOVL C01367 V=800.0 PL=0
MOVL C01368 V=800.0 PL=0
MOVL C01369 V=800.0 PL=0
MOVL C01370 V=800.0 PL=0
MOVL C01371 V=800.0 PL=0
MOVL C01372 V=800.0 PL=0
MOVL C01373 V=800.0 PL=0
MOVL C01374 V=800.0 PL=0
MOVL C01375 V=800.0 PL=0
MOVL C01376 V=800.0 PL=0
MOVL C01377 V=800.0 PL=0
MOVL C01378 V=800.0 PL=0
MOVL C01379 V=800.0 PL=0
MOVL C01380 V=800.0 PL=0
MOVL C01381 V=800.0 PL=0
MOVL C01382 V=800.0 PL=0
MOVL C01383 V=800.0 PL=0
MOVL C01384 V=800.0 PL=0
MOVL C01385 V=800.0 PL=0
MOVL C01386 V=800.0 PL=0
MOVL C01387 V=800.0 PL=0
MOVL C01388 V=800.0 PL=0
MOVL C01389 V=800.0 PL=0
MOVL C01390 V=800.0 PL=0
MOVL C01391 V=800.0 PL=0
MOVL C01392 V=800.0 PL=0
MOVL C01393 V=800.0 PL=0
MOVL C01394 V=800.0 PL=0
MOVL C01395 V=800.0 PL=0
MOVL C01396 V=800.0 PL=0
MOVL C01397 V=800.0 PL=0
MOVL C01398 V=800.0 PL=0
MOVL C01399 V=800.0 PL=0
MOVL C01400 V=800.0 PL=0
MOVL C01401 V=800.0 PL=0
MOVL C01402 V=800.0 PL=0
MOVL C01403 V=800.0 PL=0
MOVL C01404 V=800.0 PL=0
MOVL C01405 V=800.0 PL=0
MOVL C01406 V=800.0 PL=0
MOVL C01407 V=800.0 PL=0
MOVL C01408 V=800.0 PL=0
MOVL C01409 V=800.0 PL=0
MOVL C01410 V=800.0 PL=0
MOVL C01411 V=800.0 PL=0
MOVL C01412 V=800.0 PL=0
MOVL C01413 V=800.0 PL=0
MOVL C01414 V=800.0 PL=0
MOVL C01415 V=800.0 PL=0
MOVL C01416 V=800.0 PL=0
MOVL C01417 V=800.0 PL=0
MOVL C01418 V=800.0 PL=0
MOVL C01419 V=800.0 PL=0
MOVL C01420 V=800.0 PL=0
MOVL C01421 V=800.0 PL=0
MOVL C01422 V=800.0 PL=0
MOVL C01423 V=800.0 PL=0
MOVL C01424 V=800.0 PL=0
MOVL C01425 V=800.0 PL=0
MOVL C01426 V=800.0 PL=0
MOVL C01427 V=800.0 PL=0
MOVL C01428 V=800.0 PL=0
MOVL C01429 V=800.0 PL=0
MOVL C01430 V=800.0 PL=0
MOVL C01431 V=800.0 PL=0
MOVL C01432 V=800.0 PL=0
MOVL C01433 V=800.0 PL=0
MOVL C01434 V=800.0 PL=0
MOVL C01435 V=800.0 PL=0
MOVL C01436 V=800.0 PL=0
MOVL C01437 V=800.0 PL=0
MOVL C01438 V=800.0 PL=0
MOVL C01439 V=800.0 PL=0
MOVL C01440 V=800.0 PL=0
MOVL C01441 V=800.0 PL=0
MOVL C01442 V=800.0 PL=0
MOVL C01443 V=800.0 PL=0
MOVL C01444 V=800.0 PL=0
MOVL C01445 V=800.0 PL=0
MOVL C01446 V=800.0 PL=0
MOVL C01447 V=800.0 PL=0
MOVL C01448 V=800.0 PL=0
MOVL C01449 V=800.0 PL=0
MOVL C01450 V=800.0 PL=0
MOVL C01451 V=800.0 PL=0
MOVL C01452 V=800.0 PL=0
MOVL C01453 V=800.0 PL=0
MOVL C01454 V=800.0 PL=0
MOVL C01455 V=800.0 PL=0
MOVL C01456 V=800.0 PL=0
MOVL C01457 V=800.0 PL=0
MOVL C01458 V=800.0 PL=0
MOVL C01459 V=800.0 PL=0
MOVL C01460 V=800.0 PL=0
MOVL C01461 V=800.0 PL=0
MOVL C01462 V=800.0 PL=0
MOVL C01463 V=800.0 PL=0
MOVL C01464 V=800.0 PL=0
MOVL C01465 V=800.0 PL=0
MOVL C01466 V=800.0 PL=0
MOVL C01467 V=800.0 PL=0
MOVL C01468 V=800.0 PL=0
MOVL C01469 V=800.0 PL=0
MOVL C01470 V=800.0 PL=0
MOVL C01471 V=800.0 PL=0
MOVL C01472 V=800.0 PL=0
MOVL C01473 V=800.0 PL=0
MOVL C01474 V=800.0 PL=0
MOVL C01475 V=800.0 PL=0
MOVL C01476 V=800.0 PL=0
MOVL C01477 V=800.0 PL=0
MOVL C01478 V=800.0 PL=0
MOVL C01479 V=800.0 PL=0
MOVL C01480 V=800.0 PL=0
MOVL C01481 V=800.0 PL=0
MOVL C01482 V=800.0 PL=0
MOVL C01483 V=800.0 PL=0
MOVL C01484 V=800.0 PL=0
MOVL C01485 V=800.0 PL=0
MOVL C01486 V=800.0 PL=0
MOVL C01487 V=800.0 PL=0
MOVL C01488 V=800.0 PL=0
MOVL C01489 V=800.0 PL=0
MOVL C01490 V=800.0 PL=0
MOVL C01491 V=800.0 PL=0
MOVL C01492 V=800.0 PL=0
MOVL C01493 V=800.0 PL=0
MOVL C01494 V=800.0 PL=0
MOVL C01495 V=800.0 PL=0
MOVL C01496 V=800.0 PL=0
MOVL C01497 V=800.0 PL=0
MOVL C01498 V=800.0 PL=0
MOVL C01499 V=800.0 PL=0
MOVL C01500 V=800.0 PL=0
MOVL C01501 V=800.0 PL=0
MOVL C01502 V=800.0 PL=0
MOVL C01503 V=800.0 PL=0
MOVL C01504 V=800.0 PL=0
MOVL C01505 V=800.0 PL=0
MOVL C01506 V=800.0 PL=0
MOVL C01507 V=800.0 PL=0
MOVL C01508 V=800.0 PL=0
MOVL C01509 V=800.0 PL=0
MOVL C01510 V=800.0 PL=0
MOVL C01511 V=800.0 PL=0
MOVL C01512 V=800.0 PL=0
MOVL C01513 V=800.0 PL=0
MOVL C01514 V=800.0 PL=0
MOVL C01515 V=800.0 PL=0
MOVL C01516 V=800.0 PL=0
MOVL C01517 V=800.0 PL=0
MOVL C01518 V=800.0 PL=0
MOVL C01519 V=800.0 PL=0
MOVL C01520 V=800.0 PL=0
MOVL C01521 V=800.0 PL=0
MOVL C01522 V=800.0 PL=0
MOVL C01523 V=800.0 PL=0
MOVL C01524 V=800.0 PL=0
MOVL C01525 V=800.0 PL=0
MOVL C01526 V=800.0 PL=0
MOVL C01527 V=800.0 PL=0
MOVL C01528 V=800.0 PL=0
MOVL C01529 V=800.0 PL=0
MOVL C01530 V=800.0 PL=0
MOVL C01531 V=800.0 PL=0
MOVL C01532 V=800.0 PL=0
MOVL C01533 V=800.0 PL=0
MOVL C01534 V=800.0 PL=0
MOVL C01535 V=800.0 PL=0
MOVL C01536 V=800.0 PL=0
MOVL C01537 V=800.0 PL=0
MOVL C01538 V=800.0 PL=0
MOVL C01539 V=800.0 PL=0
MOVL C01540 V=800.0 PL=0
MOVL C01541 V=800.0 PL=0
MOVL C01542 V=800.0 PL=0
MOVL C01543 V=800.0 PL=0
MOVL C01544 V=800.0 PL=0
MOVL C01545 V=800.0 PL=0
MOVL C01546 V=800.0 PL=0
MOVL C01547 V=800.0 PL=0
MOVL C01548 V=800.0 PL=0
MOVL C01549 V=800.0 PL=0
MOVL C01550 V=800.0 PL=0
MOVL C01551 V=800.0 PL=0
MOVL C01552 V=800.0 PL=0
MOVL C01553 V=800.0 PL=0
MOVL C01554 V=800.0 PL=0
MOVL C01555 V=800.0 PL=0
MOVL C01556 V=800.0 PL=0
MOVL C01557 V=800.0 PL=0
MOVL C01558 V=800.0 PL=0
MOVL C01559 V=800.0 PL=0
MOVL C01560 V=800.0 PL=0
MOVL C01561 V=800.0 PL=0
MOVL C01562 V=800.0 PL=0
MOVL C01563 V=800.0 PL=0
MOVL C01564 V=800.0 PL=0
MOVL C01565 V=800.0 PL=0
MOVL C01566 V=800.0 PL=0
MOVL C01567 V=800.0 PL=0
MOVL C01568 V=800.0 PL=0
MOVL C01569 V=800.0 PL=0
MOVL C01570 V=800.0 PL=0
MOVL C01571 V=800.0 PL=0
MOVL C01572 V=800.0 PL=0
MOVL C01573 V=800.0 PL=0
MOVL C01574 V=800.0 PL=0
MOVL C01575 V=800.0 PL=0
MOVL C01576 V=800.0 PL=0
MOVL C01577 V=800.0 PL=0
MOVL C01578 V=800.0 PL=0
MOVL C01579 V=800.0 PL=0
MOVL C01580 V=800.0 PL=0
MOVL C01581 V=800.0 PL=0
MOVL C01582 V=800.0 PL=0
MOVL C01583 V=800.0 PL=0
MOVL C01584 V=800.0 PL=0
MOVL C01585 V=800.0 PL=0
MOVL C01586 V=800.0 PL=0
MOVL C01587 V=800.0 PL=0
MOVL C01588 V=800.0 PL=0
MOVL C01589 V=800.0 PL=0
MOVL C01590 V=800.0 PL=0
MOVL C01591 V=800.0 PL=0
MOVL C01592 V=800.0 PL=0
MOVL C01593 V=800.0 PL=0
MOVL C01594 V=800.0 PL=0
MOVL C01595 V=800.0 PL=0
MOVL C01596 V=800.0 PL=0
MOVL C01597 V=800.0 PL=0
MOVL C01598 V=800.0 PL=0
MOVL C01599 V=800.0 PL=0
MOVL C01600 V=800.0 PL=0
MOVL C01601 V=800.0 PL=0
MOVL C01602 V=800.0 PL=0
MOVL C01603 V=800.0 PL=0
MOVL C01604 V=800.0 PL=0
MOVL C01605 V=800.0 PL=0
MOVL C01606 V=800.0 PL=0
MOVL C01607 V=800.0 PL=0
MOVL C01608 V=800.0 PL=0
MOVL C01609 V=800.0 PL=0
MOVL C01610 V=800.0 PL=0
MOVL C01611 V=800.0 PL=0
MOVL C01612 V=800.0 PL=0
MOVL C01613 V=800.0 PL=0
MOVL C01614 V=800.0 PL=0
MOVL C01615 V=800.0 PL=0
MOVL C01616 V=800.0 PL=0
MOVL C01617 V=800.0 PL=0
MOVL C01618 V=800.0 PL=0
MOVL C01619 V=800.0 PL=0
MOVL C01620 V=800.0 PL=0
MOVL C01621 V=800.0 PL=0
MOVL C01622 V=800.0 PL=0
MOVL C01623 V=800.0 PL=0
MOVL C01624 V=800.0 PL=0
MOVL C01625 V=800.0 PL=0
MOVL C01626 V=800.0 PL=0
MOVL C01627 V=800.0 PL=0
MOVL C01628 V=800.0 PL=0
MOVL C01629 V=800.0 PL=0
MOVL C01630 V=800.0 PL=0
MOVL C01631 V=800.0 PL=0
MOVL C01632 V=800.0 PL=0
MOVL C01633 V=800.0 PL=0
MOVL C01634 V=800.0 PL=0
MOVL C01635 V=800.0 PL=0
MOVL C01636 V=800.0 PL=0
MOVL C01637 V=800.0 PL=0
MOVL C01638 V=800.0 PL=0
MOVL C01639 V=800.0 PL=0
MOVL C01640 V=800.0 PL=0
MOVL C01641 V=800.0 PL=0
MOVL C01642 V=800.0 PL=0
MOVL C01643 V=800.0 PL=0
MOVL C01644 V=800.0 PL=0
MOVL C01645 V=800.0 PL=0
MOVL C01646 V=800.0 PL=0
MOVL C01647 V=800.0 PL=0
MOVL C01648 V=800.0 PL=0
MOVL C01649 V=800.0 PL=0
MOVL C01650 V=800.0 PL=0
MOVL C01651 V=800.0 PL=0
MOVL C01652 V=800.0 PL=0
MOVL C01653 V=800.0 PL=0
MOVL C01654 V=800.0 PL=0
MOVL C01655 V=800.0 PL=0
MOVL C01656 V=800.0 PL=0
MOVL C01657 V=800.0 PL=0
MOVL C01658 V=800.0 PL=0
MOVL C01659 V=800.0 PL=0
MOVL C01660 V=800.0 PL=0
MOVL C01661 V=800.0 PL=0
MOVL C01662 V=800.0 PL=0
MOVL C01663 V=800.0 PL=0
MOVL C01664 V=800.0 PL=0
MOVL C01665 V=800.0 PL=0
MOVL C01666 V=800.0 PL=0
MOVL C01667 V=800.0 PL=0
MOVL C01668 V=800.0 PL=0
MOVL C01669 V=800.0 PL=0
MOVL C01670 V=800.0 PL=0
MOVL C01671 V=800.0 PL=0
MOVL C01672 V=800.0 PL=0
MOVL C01673 V=800.0 PL=0
MOVL C01674 V=800.0 PL=0
MOVL C01675 V=800.0 PL=0
MOVL C01676 V=800.0 PL=0
MOVL C01677 V=800.0 PL=0
MOVL C01678 V=800.0 PL=0
MOVL C01679 V=800.0 PL=0
MOVL C01680 V=800.0 PL=0
MOVL C01681 V=800.0 PL=0
MOVL C01682 V=800.0 PL=0
MOVL C01683 V=800.0 PL=0
MOVL C01684 V=800.0 PL=0
MOVL C01685 V=800.0 PL=0
MOVL C01686 V=800.0 PL=0
MOVL C01687 V=800.0 PL=0
MOVL C01688 V=800.0 PL=0
MOVL C01689 V=800.0 PL=0
MOVL C01690 V=800.0 PL=0
MOVL C01691 V=800.0 PL=0
MOVL C01692 V=800.0 PL=0
MOVL C01693 V=800.0 PL=0
MOVL C01694 V=800.0 PL=0
MOVL C01695 V=800.0 PL=0
MOVL C01696 V=800.0 PL=0
MOVL C01697 V=800.0 PL=0
MOVL C01698 V=800.0 PL=0
MOVL C01699 V=800.0 PL=0
MOVL C01700 V=800.0 PL=0
MOVL C01701 V=800.0 PL=0
MOVL C01702 V=800.0 PL=0
MOVL C01703 V=800.0 PL=0
MOVL C01704 V=800.0 PL=0
MOVL C01705 V=800.0 PL=0
MOVL C01706 V=800.0 PL=0
MOVL C01707 V=800.0 PL=0
MOVL C01708 V=800.0 PL=0
MOVL C01709 V=800.0 PL=0
MOVL C01710 V=800.0 PL=0
MOVL C01711 V=800.0 PL=0
MOVL C01712 V=800.0 PL=0
MOVL C01713 V=800.0 PL=0
MOVL C01714 V=800.0 PL=0
MOVL C01715 V=800.0 PL=0
MOVL C01716 V=800.0 PL=0
MOVL C01717 V=800.0 PL=0
MOVL C01718 V=800.0 PL=0
MOVL C01719 V=800.0 PL=0
MOVL C01720 V=800.0 PL=0
MOVL C01721 V=800.0 PL=0
MOVL C01722 V=800.0 PL=0
MOVL C01723 V=800.0 PL=0
MOVL C01724 V=800.0 PL=0
MOVL C01725 V=800.0 PL=0
MOVL C01726 V=800.0 PL=0
MOVL C01727 V=800.0 PL=0
MOVL C01728 V=800.0 PL=0
MOVL C01729 V=800.0 PL=0
MOVL C01730 V=800.0 PL=0
MOVL C01731 V=800.0 PL=0
MOVL C01732 V=800.0 PL=0
MOVL C01733 V=800.0 PL=0
MOVL C01734 V=800.0 PL=0
MOVL C01735 V=800.0 PL=0
MOVL C01736 V=800.0 PL=0
MOVL C01737 V=800.0 PL=0
MOVL C01738 V=800.0 PL=0
MOVL C01739 V=800.0 PL=0
MOVL C01740 V=800.0 PL=0
MOVL C01741 V=800.0 PL=0
MOVL C01742 V=800.0 PL=0
MOVL C01743 V=800.0 PL=0
MOVL C01744 V=800.0 PL=0
MOVL C01745 V=800.0 PL=0
MOVL C01746 V=800.0 PL=0
MOVL C01747 V=800.0 PL=0
MOVL C01748 V=800.0 PL=0
MOVL C01749 V=800.0 PL=0
MOVL C01750 V=800.0 PL=0
MOVL C01751 V=800.0 PL=0
MOVL C01752 V=800.0 PL=0
MOVL C01753 V=800.0 PL=0
MOVL C01754 V=800.0 PL=0
MOVL C01755 V=800.0 PL=0
MOVL C01756 V=800.0 PL=0
MOVL C01757 V=800.0 PL=0
MOVL C01758 V=800.0 PL=0
MOVL C01759 V=800.0 PL=0
MOVL C01760 V=800.0 PL=0
MOVL C01761 V=800.0 PL=0
MOVL C01762 V=800.0 PL=0
MOVL C01763 V=800.0 PL=0
MOVL C01764 V=800.0 PL=0
MOVL C01765 V=800.0 PL=0
MOVL C01766 V=800.0 PL=0
MOVL C01767 V=800.0 PL=0
MOVL C01768 V=800.0 PL=0
MOVL C01769 V=800.0 PL=0
MOVL C01770 V=800.0 PL=0
MOVL C01771 V=800.0 PL=0
MOVL C01772 V=800.0 PL=0
MOVL C01773 V=800.0 PL=0
MOVL C01774 V=800.0 PL=0
MOVL C01775 V=800.0 PL=0
MOVL C01776 V=800.0 PL=0
MOVL C01777 V=800.0 PL=0
MOVL C01778 V=800.0 PL=0
MOVL C01779 V=800.0 PL=0
MOVL C01780 V=800.0 PL=0
MOVL C01781 V=800.0 PL=0
MOVL C01782 V=800.0 PL=0
MOVL C01783 V=800.0 PL=0
MOVL C01784 V=800.0 PL=0
MOVL C01785 V=800.0 PL=0
MOVL C01786 V=800.0 PL=0
MOVL C01787 V=800.0 PL=0
MOVL C01788 V=800.0 PL=0
MOVL C01789 V=800.0 PL=0
MOVL C01790 V=800.0 PL=0
MOVL C01791 V=800.0 PL=0
MOVL C01792 V=800.0 PL=0
MOVL C01793 V=800.0 PL=0
MOVL C01794 V=800.0 PL=0
MOVL C01795 V=800.0 PL=0
MOVL C01796 V=800.0 PL=0
MOVL C01797 V=800.0 PL=0
MOVL C01798 V=800.0 PL=0
MOVL C01799 V=800.0 PL=0
MOVL C01800 V=800.0 PL=0
MOVL C01801 V=800.0 PL=0
MOVL C01802 V=800.0 PL=0
MOVL C01803 V=800.0 PL=0
MOVL C01804 V=800.0 PL=0
MOVL C01805 V=800.0 PL=0
MOVL C01806 V=800.0 PL=0
MOVL C01807 V=800.0 PL=0
MOVL C01808 V=800.0 PL=0
MOVL C01809 V=800.0 PL=0
MOVL C01810 V=800.0 PL=0
MOVL C01811 V=800.0 PL=0
MOVL C01812 V=800.0 PL=0
MOVL C01813 V=800.0 PL=0
MOVL C01814 V=800.0 PL=0
MOVL C01815 V=800.0 PL=0
MOVL C01816 V=800.0 PL=0
MOVL C01817 V=800.0 PL=0
MOVL C01818 V=800.0 PL=0
MOVL C01819 V=800.0 PL=0
MOVL C01820 V=800.0 PL=0
MOVL C01821 V=800.0 PL=0
MOVL C01822 V=800.0 PL=0
MOVL C01823 V=800.0 PL=0
MOVL C01824 V=800.0 PL=0
MOVL C01825 V=800.0 PL=0
MOVL C01826 V=800.0 PL=0
MOVL C01827 V=800.0 PL=0
MOVL C01828 V=800.0 PL=0
MOVL C01829 V=800.0 PL=0
MOVL C01830 V=800.0 PL=0
MOVL C01831 V=800.0 PL=0
MOVL C01832 V=800.0 PL=0
MOVL C01833 V=800.0 PL=0
MOVL C01834 V=800.0 PL=0
MOVL C01835 V=800.0 PL=0
MOVL C01836 V=800.0 PL=0
MOVL C01837 V=800.0 PL=0
MOVL C01838 V=800.0 PL=0
MOVL C01839 V=800.0 PL=0
MOVL C01840 V=800.0 PL=0
MOVL C01841 V=800.0 PL=0
MOVL C01842 V=800.0 PL=0
MOVL C01843 V=800.0 PL=0
MOVL C01844 V=800.0 PL=0
MOVL C01845 V=800.0 PL=0
MOVL C01846 V=800.0 PL=0
MOVL C01847 V=800.0 PL=0
MOVL C01848 V=800.0 PL=0
MOVL C01849 V=800.0 PL=0
MOVL C01850 V=800.0 PL=0
MOVL C01851 V=800.0 PL=0
MOVL C01852 V=800.0 PL=0
MOVL C01853 V=800.0 PL=0
MOVL C01854 V=800.0 PL=0
MOVL C01855 V=800.0 PL=0
MOVL C01856 V=800.0 PL=0
MOVL C01857 V=800.0 PL=0
MOVL C01858 V=800.0 PL=0
MOVL C01859 V=800.0 PL=0
MOVL C01860 V=800.0 PL=0
MOVL C01861 V=800.0 PL=0
MOVL C01862 V=800.0 PL=0
MOVL C01863 V=800.0 PL=0
MOVL C01864 V=800.0 PL=0
MOVL C01865 V=800.0 PL=0
MOVL C01866 V=800.0 PL=0
MOVL C01867 V=800.0 PL=0
MOVL C01868 V=800.0 PL=0
MOVL C01869 V=800.0 PL=0
MOVL C01870 V=800.0 PL=0
MOVL C01871 V=800.0 PL=0
MOVL C01872 V=800.0 PL=0
MOVL C01873 V=800.0 PL=0
MOVL C01874 V=800.0 PL=0
MOVL C01875 V=800.0 PL=0
MOVL C01876 V=800.0 PL=0
MOVL C01877 V=800.0 PL=0
MOVL C01878 V=800.0 PL=0
MOVL C01879 V=800.0 PL=0
MOVL C01880 V=800.0 PL=0
MOVL C01881 V=800.0 PL=0
MOVL C01882 V=800.0 PL=0
MOVL C01883 V=800.0 PL=0
MOVL C01884 V=800.0 PL=0
MOVL C01885 V=800.0 PL=0
MOVL C01886 V=800.0 PL=0
MOVL C01887 V=800.0 PL=0
MOVL C01888 V=800.0 PL=0
MOVL C01889 V=800.0 PL=0
MOVL C01890 V=800.0 PL=0
MOVL C01891 V=800.0 PL=0
MOVL C01892 V=800.0 PL=0
MOVL C01893 V=800.0 PL=0
MOVL C01894 V=800.0 PL=0
MOVL C01895 V=800.0 PL=0
MOVL C01896 V=800.0 PL=0
MOVL C01897 V=800.0 PL=0
MOVL C01898 V=800.0 PL=0
MOVL C01899 V=800.0 PL=0
MOVL C01900 V=800.0 PL=0
MOVL C01901 V=800.0 PL=0
MOVL C01902 V=800.0 PL=0
MOVL C01903 V=800.0 PL=0
MOVL C01904 V=800.0 PL=0
MOVL C01905 V=800.0 PL=0
MOVL C01906 V=800.0 PL=0
MOVL C01907 V=800.0 PL=0
MOVL C01908 V=800.0 PL=0
MOVL C01909 V=800.0 PL=0
MOVL C01910 V=800.0 PL=0
MOVL C01911 V=800.0 PL=0
MOVL C01912 V=800.0 PL=0
MOVL C01913 V=800.0 PL=0
MOVL C01914 V=800.0 PL=0
MOVL C01915 V=800.0 PL=0
MOVL C01916 V=800.0 PL=0
MOVL C01917 V=800.0 PL=0
MOVL C01918 V=800.0 PL=0
MOVL C01919 V=800.0 PL=0
MOVL C01920 V=800.0 PL=0
MOVL C01921 V=800.0 PL=0
MOVL C01922 V=800.0 PL=0
MOVL C01923 V=800.0 PL=0
MOVL C01924 V=800.0 PL=0
MOVL C01925 V=800.0 PL=0
MOVL C01926 V=800.0 PL=0
MOVL C01927 V=800.0 PL=0
MOVL C01928 V=800.0 PL=0
MOVL C01929 V=800.0 PL=0
MOVL C01930 V=800.0 PL=0
MOVL C01931 V=800.0 PL=0
MOVL C01932 V=800.0 PL=0
MOVL C01933 V=800.0 PL=0
MOVL C01934 V=800.0 PL=0
MOVL C01935 V=800.0 PL=0
MOVL C01936 V=800.0 PL=0
MOVL C01937 V=800.0 PL=0
MOVL C01938 V=800.0 PL=0
MOVL C01939 V=800.0 PL=0
MOVL C01940 V=800.0 PL=0
MOVL C01941 V=800.0 PL=0
MOVL C01942 V=800.0 PL=0
MOVL C01943 V=800.0 PL=0
MOVL C01944 V=800.0 PL=0
MOVL C01945 V=800.0 PL=0
MOVL C01946 V=800.0 PL=0
MOVL C01947 V=800.0 PL=0
MOVL C01948 V=800.0 PL=0
MOVL C01949 V=800.0 PL=0
MOVL C01950 V=800.0 PL=0
MOVL C01951 V=800.0 PL=0
MOVL C01952 V=800.0 PL=0
MOVL C01953 V=800.0 PL=0
MOVL C01954 V=800.0 PL=0
MOVL C01955 V=800.0 PL=0
MOVL C01956 V=800.0 PL=0
MOVL C01957 V=800.0 PL=0
MOVL C01958 V=800.0 PL=0
MOVL C01959 V=800.0 PL=0
MOVL C01960 V=800.0 PL=0
MOVL C01961 V=800.0 PL=0
MOVL C01962 V=800.0 PL=0
MOVL C01963 V=800.0 PL=0
MOVL C01964 V=800.0 PL=0
MOVL C01965 V=800.0 PL=0
MOVL C01966 V=800.0 PL=0
MOVL C01967 V=800.0 PL=0
MOVL C01968 V=800.0 PL=0
MOVL C01969 V=800.0 PL=0
MOVL C01970 V=800.0 PL=0
MOVL C01971 V=800.0 PL=0
MOVL C01972 V=800.0 PL=0
MOVL C01973 V=800.0 PL=0
MOVL C01974 V=800.0 PL=0
MOVL C01975 V=800.0 PL=0
MOVL C01976 V=800.0 PL=0
MOVL C01977 V=800.0 PL=0
MOVL C01978 V=800.0 PL=0
MOVL C01979 V=800.0 PL=0
MOVL C01980 V=800.0 PL=0
MOVL C01981 V=800.0 PL=0
MOVL C01982 V=800.0 PL=0
MOVL C01983 V=800.0 PL=0
MOVL C01984 V=800.0 PL=0
MOVL C01985 V=800.0 PL=0
MOVL C01986 V=800.0 PL=0
MOVL C01987 V=800.0 PL=0
MOVL C01988 V=800.0 PL=0
MOVL C01989 V=800.0 PL=0
MOVL C01990 V=800.0 PL=0
MOVL C01991 V=800.0 PL=0
MOVL C01992 V=800.0 PL=0
MOVL C01993 V=800.0 PL=0
MOVL C01994 V=800.0 PL=0
MOVL C01995 V=800.0 PL=0
MOVL C01996 V=800.0 PL=0
MOVL C01997 V=800.0 PL=0
MOVL C01998 V=800.0 PL=0
MOVL C01999 V=800.0 PL=0
MOVL C02000 V=800.0 PL=0
MOVL C02001 V=800.0 PL=0
MOVL C02002 V=800.0 PL=0
MOVL C02003 V=800.0 PL=0
MOVL C02004 V=800.0 PL=0
MOVL C02005 V=800.0 PL=0
MOVL C02006 V=800.0 PL=0
MOVL C02007 V=800.0 PL=0
MOVL C02008 V=800.0 PL=0
MOVL C02009 V=800.0 PL=0
MOVL C02010 V=800.0 PL=0
MOVL C02011 V=800.0 PL=0
MOVL C02012 V=800.0 PL=0
MOVL C02013 V=800.0 PL=0
MOVL C02014 V=800.0 PL=0
MOVL C02015 V=800.0 PL=0
MOVL C02016 V=800.0 PL=0
MOVL C02017 V=800.0 PL=0
MOVL C02018 V=800.0 PL=0
MOVL C02019 V=800.0 PL=0
MOVL C02020 V=800.0 PL=0
MOVL C02021 V=800.0 PL=0
MOVL C02022 V=800.0 PL=0
MOVL C02023 V=800.0 PL=0
MOVL C02024 V=800.0 PL=0
MOVL C02025 V=800.0 PL=0
MOVL C02026 V=800.0 PL=0
MOVL C02027 V=800.0 PL=0
MOVL C02028 V=800.0 PL=0
MOVL C02029 V=800.0 PL=0
MOVL C02030 V=800.0 PL=0
MOVL C02031 V=800.0 PL=0
MOVL C02032 V=800.0 PL=0
MOVL C02033 V=800.0 PL=0
MOVL C02034 V=800.0 PL=0
MOVL C02035 V=800.0 PL=0
MOVL C02036 V=800.0 PL=0
MOVL C02037 V=800.0 PL=0
